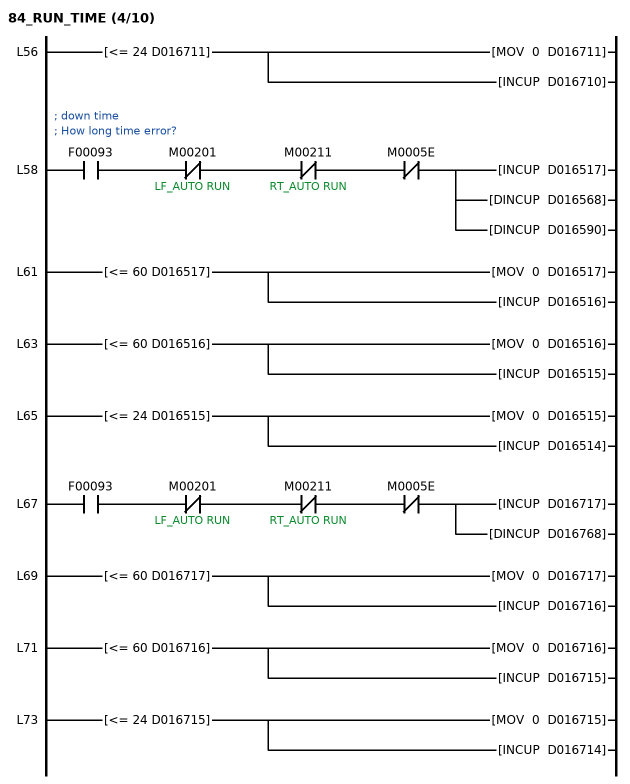
[picture p360: 84_RUN_TIME rungs L56-L73]
; L56
LOAD<=    24 D016711
MOV       0 D016711
INCUP     D016710
; L58
LOAD      F00093
AND NOT   M00201	// LF_AUTO RUN
AND NOT   M00211	// RT_AUTO RUN
AND NOT   M0005E
INCUP     D016517
DINCUP    D016568
DINCUP    D016590
// output comment: down time
// output comment: How long time error?
; L61
LOAD<=    60 D016517
MOV       0 D016517
INCUP     D016516
; L63
LOAD<=    60 D016516
MOV       0 D016516
INCUP     D016515
; L65
LOAD<=    24 D016515
MOV       0 D016515
INCUP     D016514
; L67
LOAD      F00093
AND NOT   M00201	// LF_AUTO RUN
AND NOT   M00211	// RT_AUTO RUN
AND NOT   M0005E
INCUP     D016717
DINCUP    D016768
; L69
LOAD<=    60 D016717
MOV       0 D016717
INCUP     D016716
; L71
LOAD<=    60 D016716
MOV       0 D016716
INCUP     D016715
; L73
LOAD<=    24 D016715
MOV       0 D016715
INCUP     D016714

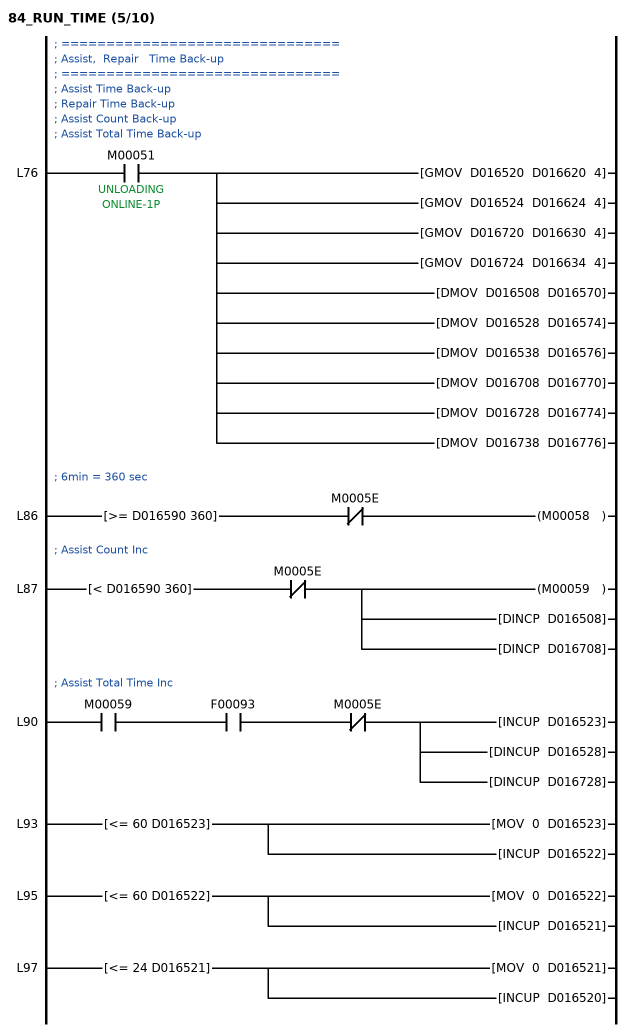
// ===============================
// Assist,  Repair   Time Back-up
// ===============================
; L76
LOAD      M00051	// UNLOADING ONLINE-1P
GMOV      D016520 D016620 4
GMOV      D016524 D016624 4
GMOV      D016720 D016630 4
GMOV      D016724 D016634 4
DMOV      D016508 D016570
DMOV      D016528 D016574
DMOV      D016538 D016576
DMOV      D016708 D016770
DMOV      D016728 D016774
DMOV      D016738 D016776
// output comment: Assist Time Back-up
// output comment: Repair Time Back-up
// output comment: Assist Count Back-up
// output comment: Assist Total Time Back-up
; L86
LOAD>=    D016590 360
AND NOT   M0005E
OUT       M00058
// output comment: 6min = 360 sec
; L87
LOAD<     D016590 360
AND NOT   M0005E
OUT       M00059
DINCP     D016508
DINCP     D016708
// output comment: Assist Count Inc
; L90
LOAD      M00059
AND       F00093
AND NOT   M0005E
INCUP     D016523
DINCUP    D016528
DINCUP    D016728
// output comment: Assist Total Time Inc
; L93
LOAD<=    60 D016523
MOV       0 D016523
INCUP     D016522
; L95
LOAD<=    60 D016522
MOV       0 D016522
INCUP     D016521
; L97
LOAD<=    24 D016521
MOV       0 D016521
INCUP     D016520

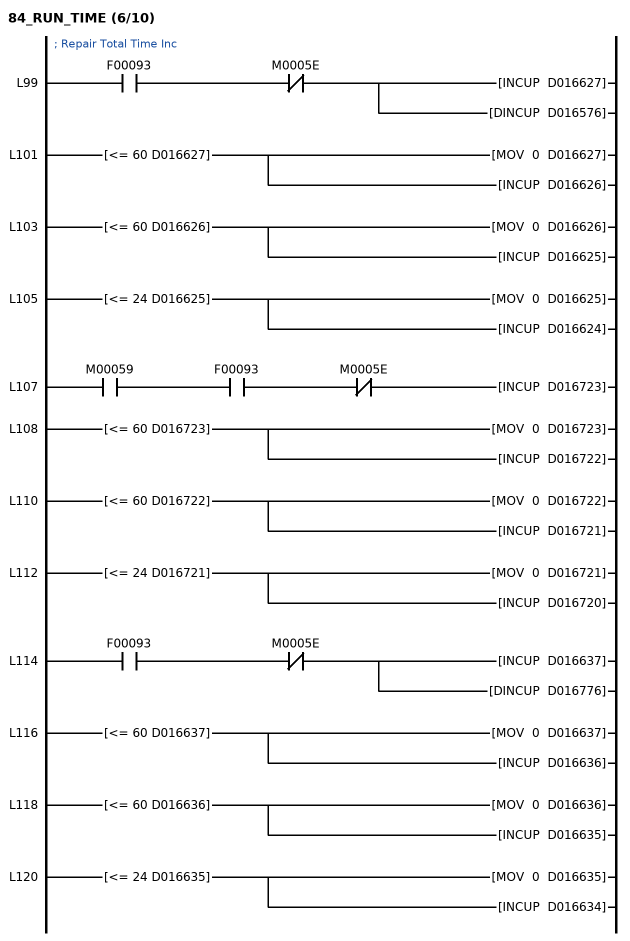
; L99
LOAD      F00093
AND NOT   M0005E
INCUP     D016627
DINCUP    D016576
// output comment: Repair Total Time Inc
; L101
LOAD<=    60 D016627
MOV       0 D016627
INCUP     D016626
; L103
LOAD<=    60 D016626
MOV       0 D016626
INCUP     D016625
; L105
LOAD<=    24 D016625
MOV       0 D016625
INCUP     D016624
; L107
LOAD      M00059
AND       F00093
AND NOT   M0005E
INCUP     D016723
; L108
LOAD<=    60 D016723
MOV       0 D016723
INCUP     D016722
; L110
LOAD<=    60 D016722
MOV       0 D016722
INCUP     D016721
; L112
LOAD<=    24 D016721
MOV       0 D016721
INCUP     D016720
; L114
LOAD      F00093
AND NOT   M0005E
INCUP     D016637
DINCUP    D016776
; L116
LOAD<=    60 D016637
MOV       0 D016637
INCUP     D016636
; L118
LOAD<=    60 D016636
MOV       0 D016636
INCUP     D016635
; L120
LOAD<=    24 D016635
MOV       0 D016635
INCUP     D016634

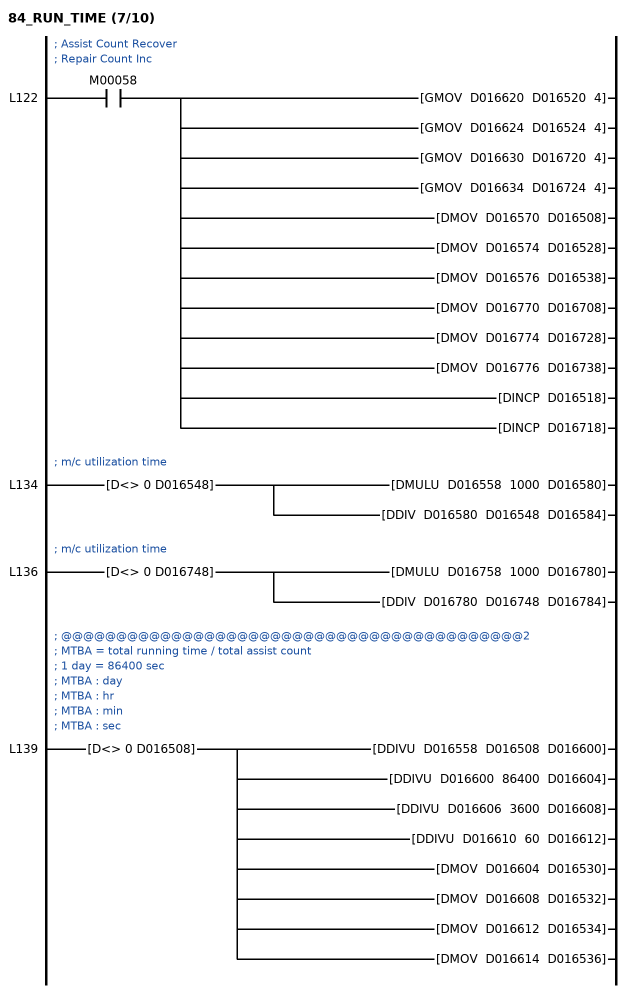
; L122
LOAD      M00058
GMOV      D016620 D016520 4
GMOV      D016624 D016524 4
GMOV      D016630 D016720 4
GMOV      D016634 D016724 4
DMOV      D016570 D016508
DMOV      D016574 D016528
DMOV      D016576 D016538
DMOV      D016770 D016708
DMOV      D016774 D016728
DMOV      D016776 D016738
DINCP     D016518
DINCP     D016718
// output comment: Assist Count Recover
// output comment: Repair Count Inc
; L134
LOADD<>   0 D016548
DMULU     D016558 1000 D016580
DDIV      D016580 D016548 D016584
// output comment: m/c utilization time
; L136
LOADD<>   0 D016748
DMULU     D016758 1000 D016780
DDIV      D016780 D016748 D016784
// output comment: m/c utilization time
// @@@@@@@@@@@@@@@@@@@@@@@@@@@@@@@@@@@@@@@@@@2
; L139
LOADD<>   0 D016508
DDIVU     D016558 D016508 D016600
DDIVU     D016600 86400 D016604
DDIVU     D016606 3600 D016608
DDIVU     D016610 60 D016612
DMOV      D016604 D016530
DMOV      D016608 D016532
DMOV      D016612 D016534
DMOV      D016614 D016536
// output comment: MTBA = total running time / total assist count
// output comment: 1 day = 86400 sec
// output comment: MTBA : day
// output comment: MTBA : hr
// output comment: MTBA : min
// output comment: MTBA : sec

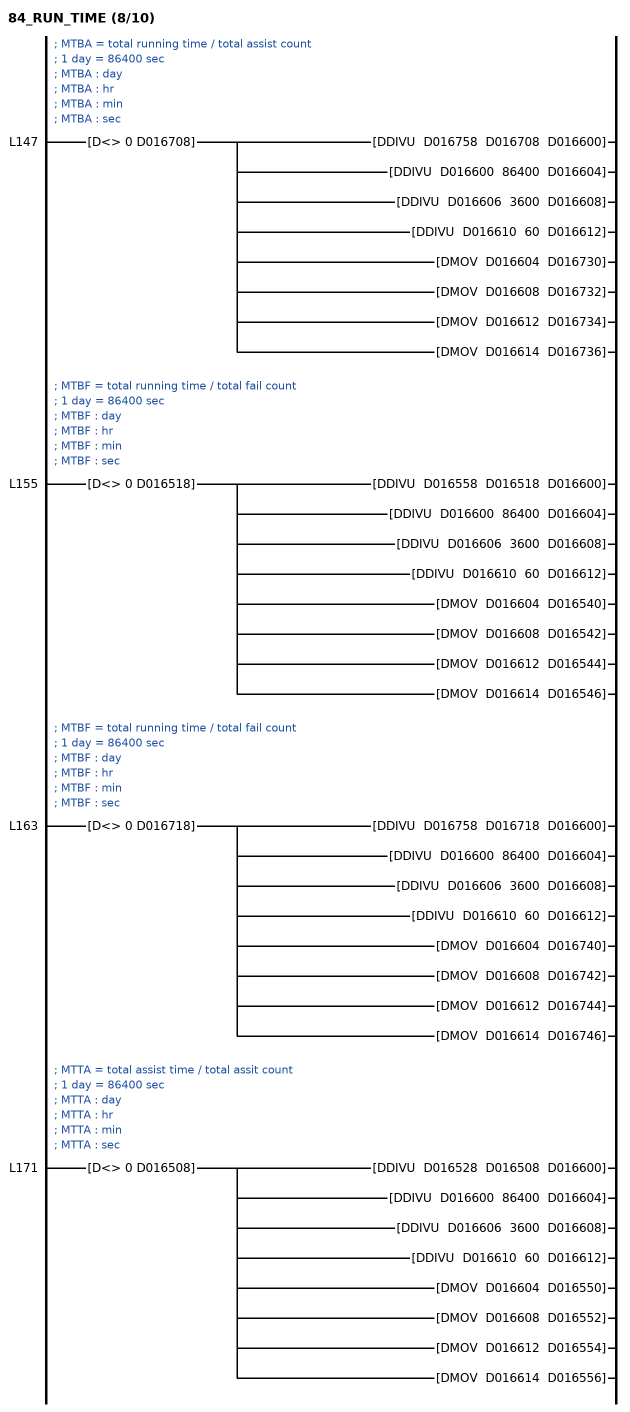
; L147
LOADD<>   0 D016708
DDIVU     D016758 D016708 D016600
DDIVU     D016600 86400 D016604
DDIVU     D016606 3600 D016608
DDIVU     D016610 60 D016612
DMOV      D016604 D016730
DMOV      D016608 D016732
DMOV      D016612 D016734
DMOV      D016614 D016736
// output comment: MTBA = total running time / total assist count
// output comment: 1 day = 86400 sec
// output comment: MTBA : day
// output comment: MTBA : hr
// output comment: MTBA : min
// output comment: MTBA : sec
; L155
LOADD<>   0 D016518
DDIVU     D016558 D016518 D016600
DDIVU     D016600 86400 D016604
DDIVU     D016606 3600 D016608
DDIVU     D016610 60 D016612
DMOV      D016604 D016540
DMOV      D016608 D016542
DMOV      D016612 D016544
DMOV      D016614 D016546
// output comment: MTBF = total running time / total fail count
// output comment: 1 day = 86400 sec
// output comment: MTBF : day
// output comment: MTBF : hr
// output comment: MTBF : min
// output comment: MTBF : sec
; L163
LOADD<>   0 D016718
DDIVU     D016758 D016718 D016600
DDIVU     D016600 86400 D016604
DDIVU     D016606 3600 D016608
DDIVU     D016610 60 D016612
DMOV      D016604 D016740
DMOV      D016608 D016742
DMOV      D016612 D016744
DMOV      D016614 D016746
// output comment: MTBF = total running time / total fail count
// output comment: 1 day = 86400 sec
// output comment: MTBF : day
// output comment: MTBF : hr
// output comment: MTBF : min
// output comment: MTBF : sec
; L171
LOADD<>   0 D016508
DDIVU     D016528 D016508 D016600
DDIVU     D016600 86400 D016604
DDIVU     D016606 3600 D016608
DDIVU     D016610 60 D016612
DMOV      D016604 D016550
DMOV      D016608 D016552
DMOV      D016612 D016554
DMOV      D016614 D016556
// output comment: MTTA = total assist time / total assit count
// output comment: 1 day = 86400 sec
// output comment: MTTA : day
// output comment: MTTA : hr
// output comment: MTTA : min
// output comment: MTTA : sec

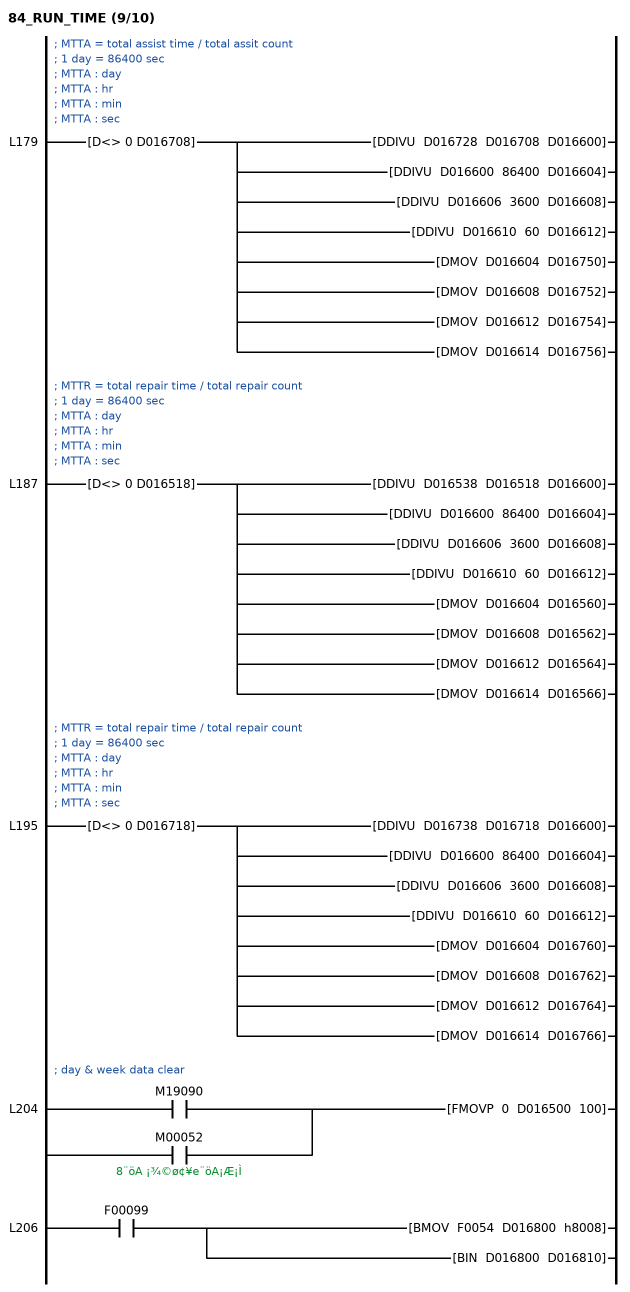
; L179
LOADD<>   0 D016708
DDIVU     D016728 D016708 D016600
DDIVU     D016600 86400 D016604
DDIVU     D016606 3600 D016608
DDIVU     D016610 60 D016612
DMOV      D016604 D016750
DMOV      D016608 D016752
DMOV      D016612 D016754
DMOV      D016614 D016756
// output comment: MTTA = total assist time / total assit count
// output comment: 1 day = 86400 sec
// output comment: MTTA : day
// output comment: MTTA : hr
// output comment: MTTA : min
// output comment: MTTA : sec
; L187
LOADD<>   0 D016518
DDIVU     D016538 D016518 D016600
DDIVU     D016600 86400 D016604
DDIVU     D016606 3600 D016608
DDIVU     D016610 60 D016612
DMOV      D016604 D016560
DMOV      D016608 D016562
DMOV      D016612 D016564
DMOV      D016614 D016566
// output comment: MTTR = total repair time / total repair count
// output comment: 1 day = 86400 sec
// output comment: MTTA : day
// output comment: MTTA : hr
// output comment: MTTA : min
// output comment: MTTA : sec
; L195
LOADD<>   0 D016718
DDIVU     D016738 D016718 D016600
DDIVU     D016600 86400 D016604
DDIVU     D016606 3600 D016608
DDIVU     D016610 60 D016612
DMOV      D016604 D016760
DMOV      D016608 D016762
DMOV      D016612 D016764
DMOV      D016614 D016766
// output comment: MTTR = total repair time / total repair count
// output comment: 1 day = 86400 sec
// output comment: MTTA : day
// output comment: MTTA : hr
// output comment: MTTA : min
// output comment: MTTA : sec
// day & week data clear
; L204
LOAD      M19090
OR        M00052	// 8¨öA ¡¾©ø¢¥e¨öA¡Æ¡Ì
FMOVP     0 D016500 100
; L206
LOAD      F00099
BMOV      F0054 D016800 h8008
BIN       D016800 D016810

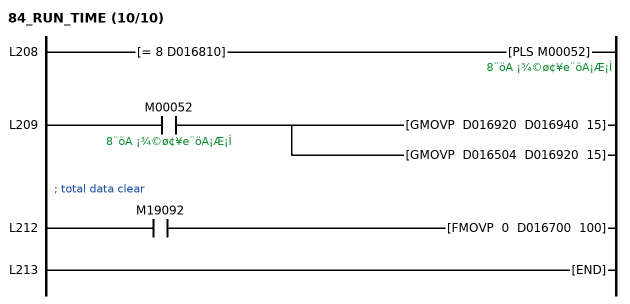
; L208
LOAD=     8 D016810
OUTP      M00052	// 8¨öA ¡¾©ø¢¥e¨öA¡Æ¡Ì
; L209
LOAD      M00052	// 8¨öA ¡¾©ø¢¥e¨öA¡Æ¡Ì
GMOVP     D016920 D016940 15
GMOVP     D016504 D016920 15
// total data clear
; L212
LOAD      M19092
FMOVP     0 D016700 100
; L213
END

PROGRAM 90_ALARM (task: ¨ö¨¬A¥ì CA¡¤I¡¾¡¿¡¤¡Í)

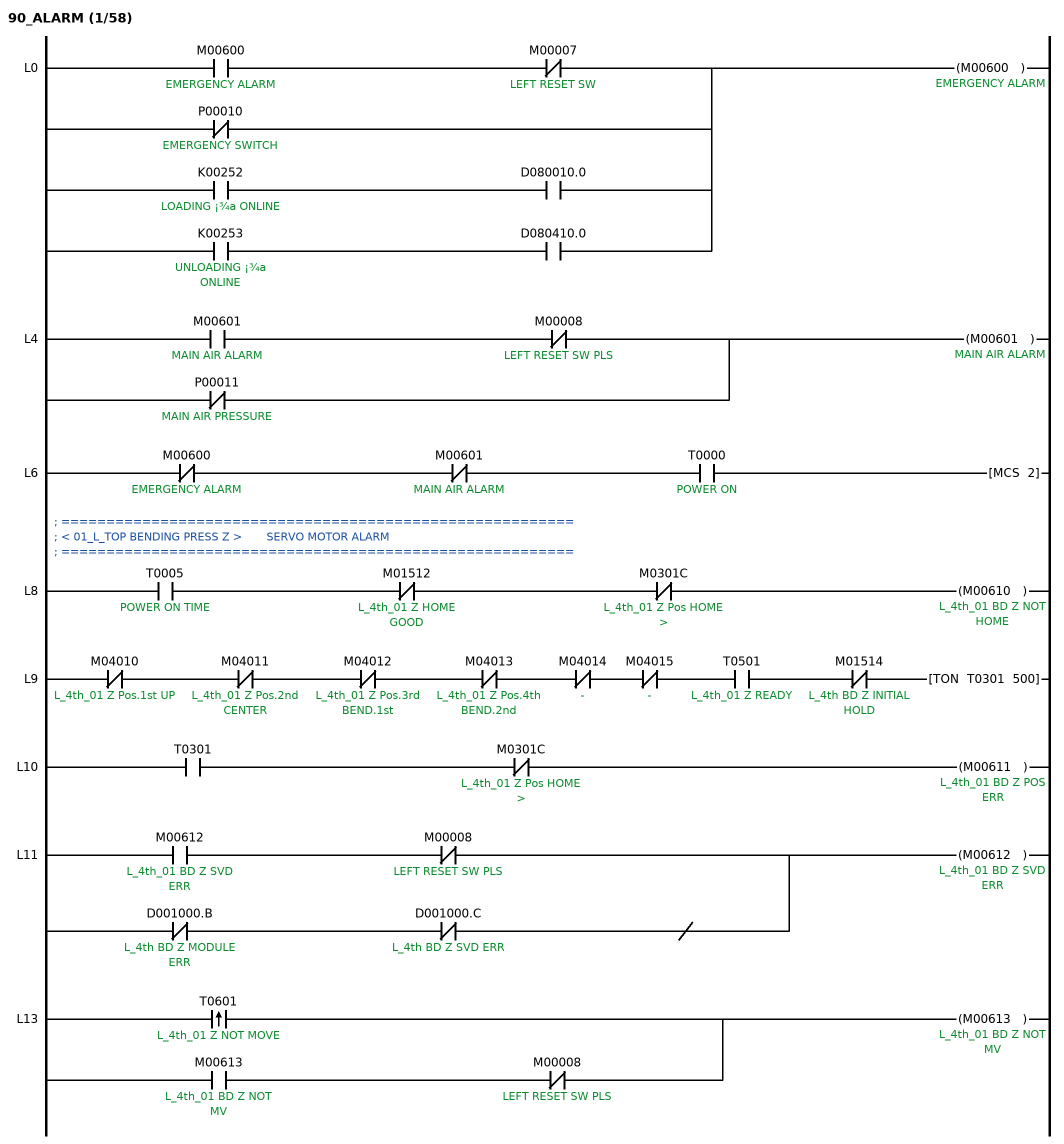
; L0
LOAD      M00600	// EMERGENCY ALARM
AND NOT   M00007	// LEFT RESET SW
OR NOT    P00010	// EMERGENCY SWITCH
LOAD      K00252	// LOADING ¡¾a ONLINE
AND       D080010.0
OR LOAD
LOAD      K00253	// UNLOADING ¡¾a ONLINE
AND       D080410.0
OR LOAD
OUT       M00600	// EMERGENCY ALARM
; L4
LOAD      M00601	// MAIN AIR ALARM
AND NOT   M00008	// LEFT RESET SW PLS
OR NOT    P00011	// MAIN AIR PRESSURE
OUT       M00601	// MAIN AIR ALARM
; L6
LOAD NOT  M00600	// EMERGENCY ALARM
AND NOT   M00601	// MAIN AIR ALARM
AND       T0000	// POWER ON
MCS       2
// =========================================================
// 
//        < 01_L_TOP BENDING PRESS Z >       SERVO MOTOR ALARM
// 
// =========================================================
; L8
LOAD      T0005	// POWER ON TIME
AND NOT   M01512	// L_4th_01 Z HOME GOOD
AND NOT   M0301C	// L_4th_01 Z Pos HOME >
OUT       M00610	// L_4th_01 BD Z NOT HOME
; L9
LOAD NOT  M04010	// L_4th_01 Z Pos.1st UP
AND NOT   M04011	// L_4th_01 Z Pos.2nd CENTER
AND NOT   M04012	// L_4th_01 Z Pos.3rd BEND.1st
AND NOT   M04013	// L_4th_01 Z Pos.4th BEND.2nd
AND NOT   M04014	// -
AND NOT   M04015	// -
AND       T0501	// L_4th_01 Z READY
AND NOT   M01514	// L_4th BD Z INITIAL HOLD
TON       T0301 500
; L10
LOAD      T0301
AND NOT   M0301C	// L_4th_01 Z Pos HOME >
OUT       M00611	// L_4th_01 BD Z POS ERR
; L11
LOAD      M00612	// L_4th_01 BD Z SVD ERR
AND NOT   M00008	// LEFT RESET SW PLS
LOAD NOT  D001000.B	// L_4th BD Z MODULE ERR
AND NOT   D001000.C	// L_4th BD Z SVD ERR
NOT
OR LOAD
OUT       M00612	// L_4th_01 BD Z SVD ERR
; L13
LOADP     T0601	// L_4th_01 Z NOT MOVE
LOAD      M00613	// L_4th_01 BD Z NOT MV
AND NOT   M00008	// LEFT RESET SW PLS
OR LOAD
OUT       M00613	// L_4th_01 BD Z NOT MV

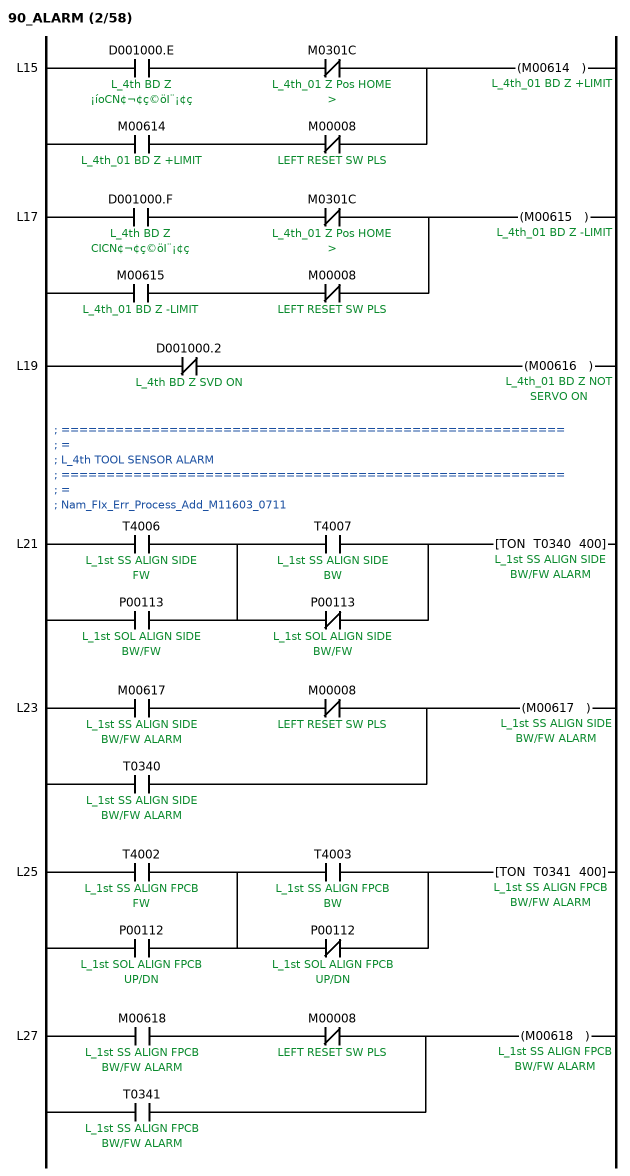
; L15
LOAD      D001000.E	// L_4th BD Z ¡íoCN¢¬¢ç©öI¨¡¢ç
AND NOT   M0301C	// L_4th_01 Z Pos HOME >
LOAD      M00614	// L_4th_01 BD Z +LIMIT
AND NOT   M00008	// LEFT RESET SW PLS
OR LOAD
OUT       M00614	// L_4th_01 BD Z +LIMIT
; L17
LOAD      D001000.F	// L_4th BD Z CICN¢¬¢ç©öI¨¡¢ç
AND NOT   M0301C	// L_4th_01 Z Pos HOME >
LOAD      M00615	// L_4th_01 BD Z -LIMIT
AND NOT   M00008	// LEFT RESET SW PLS
OR LOAD
OUT       M00615	// L_4th_01 BD Z -LIMIT
; L19
LOAD NOT  D001000.2	// L_4th BD Z SVD ON
OUT       M00616	// L_4th_01 BD Z NOT SERVO ON
// =========================================================
// 
//        L_4th TOOL SENSOR ALARM
// 
// =========================================================
; L21
LOAD      T4006	// L_1st SS ALIGN SIDE FW
OR        P00113	// L_1st SOL ALIGN SIDE BW/FW
LOAD      T4007	// L_1st SS ALIGN SIDE BW
OR NOT    P00113	// L_1st SOL ALIGN SIDE BW/FW
AND LOAD
TON       T0340 400	// L_1st SS ALIGN SIDE BW/FW ALARM
// output comment: Nam_FIx_Err_Process_Add_M11603_0711
; L23
LOAD      M00617	// L_1st SS ALIGN SIDE BW/FW ALARM
AND NOT   M00008	// LEFT RESET SW PLS
OR        T0340	// L_1st SS ALIGN SIDE BW/FW ALARM
OUT       M00617	// L_1st SS ALIGN SIDE BW/FW ALARM
; L25
LOAD      T4002	// L_1st SS ALIGN FPCB FW
OR        P00112	// L_1st SOL ALIGN FPCB UP/DN
LOAD      T4003	// L_1st SS ALIGN FPCB BW
OR NOT    P00112	// L_1st SOL ALIGN FPCB UP/DN
AND LOAD
TON       T0341 400	// L_1st SS ALIGN FPCB BW/FW ALARM
; L27
LOAD      M00618	// L_1st SS ALIGN FPCB BW/FW ALARM
AND NOT   M00008	// LEFT RESET SW PLS
OR        T0341	// L_1st SS ALIGN FPCB BW/FW ALARM
OUT       M00618	// L_1st SS ALIGN FPCB BW/FW ALARM

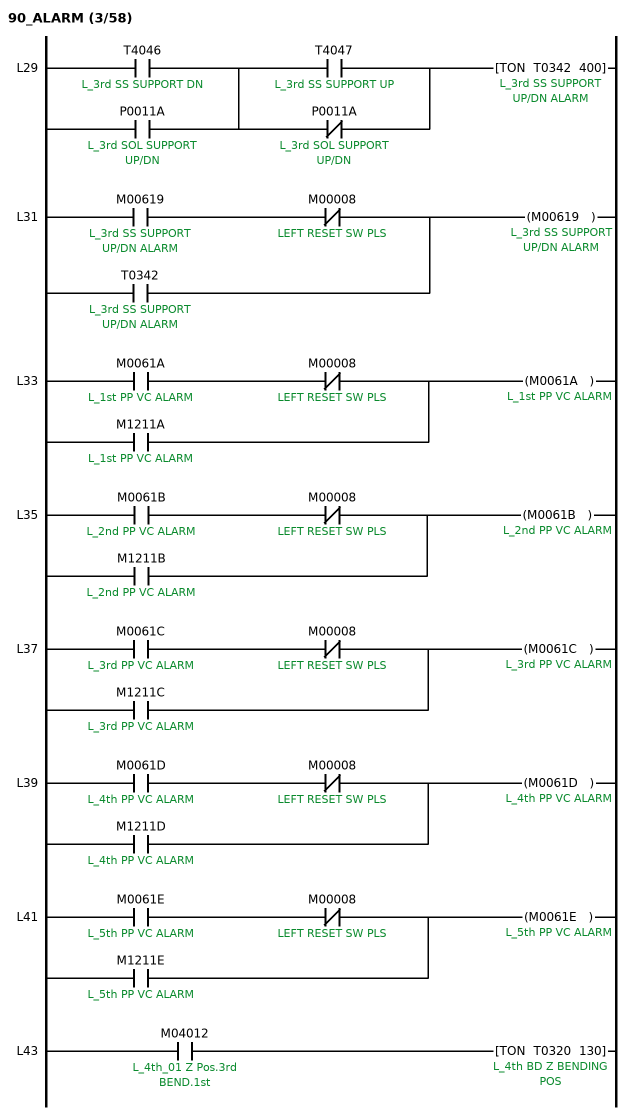
; L29
LOAD      T4046	// L_3rd SS SUPPORT DN
OR        P0011A	// L_3rd SOL SUPPORT UP/DN
LOAD      T4047	// L_3rd SS SUPPORT UP
OR NOT    P0011A	// L_3rd SOL SUPPORT UP/DN
AND LOAD
TON       T0342 400	// L_3rd SS SUPPORT UP/DN ALARM
; L31
LOAD      M00619	// L_3rd SS SUPPORT UP/DN ALARM
AND NOT   M00008	// LEFT RESET SW PLS
OR        T0342	// L_3rd SS SUPPORT UP/DN ALARM
OUT       M00619	// L_3rd SS SUPPORT UP/DN ALARM
; L33
LOAD      M0061A	// L_1st PP VC ALARM
AND NOT   M00008	// LEFT RESET SW PLS
OR        M1211A	// L_1st PP VC ALARM
OUT       M0061A	// L_1st PP VC ALARM
; L35
LOAD      M0061B	// L_2nd PP VC ALARM
AND NOT   M00008	// LEFT RESET SW PLS
OR        M1211B	// L_2nd PP VC ALARM
OUT       M0061B	// L_2nd PP VC ALARM
; L37
LOAD      M0061C	// L_3rd PP VC ALARM
AND NOT   M00008	// LEFT RESET SW PLS
OR        M1211C	// L_3rd PP VC ALARM
OUT       M0061C	// L_3rd PP VC ALARM
; L39
LOAD      M0061D	// L_4th PP VC ALARM
AND NOT   M00008	// LEFT RESET SW PLS
OR        M1211D	// L_4th PP VC ALARM
OUT       M0061D	// L_4th PP VC ALARM
; L41
LOAD      M0061E	// L_5th PP VC ALARM
AND NOT   M00008	// LEFT RESET SW PLS
OR        M1211E	// L_5th PP VC ALARM
OUT       M0061E	// L_5th PP VC ALARM
; L43
LOAD      M04012	// L_4th_01 Z Pos.3rd BEND.1st
TON       T0320 130	// L_4th BD Z BENDING POS

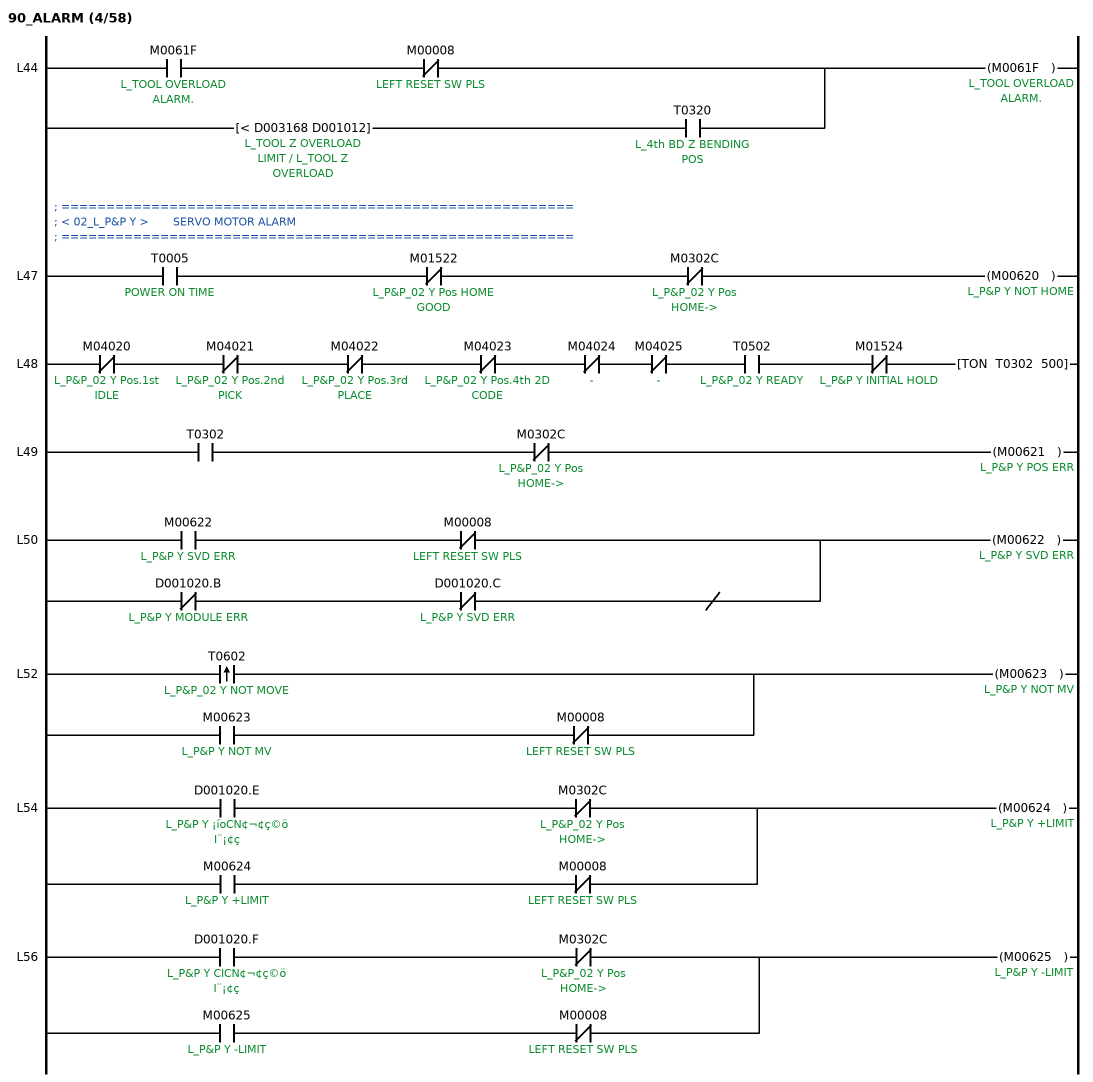
; L44
LOAD      M0061F	// L_TOOL OVERLOAD ALARM.
AND NOT   M00008	// LEFT RESET SW PLS
LOAD<     D003168 D001012	// L_TOOL Z OVERLOAD LIMIT / L_TOOL Z OVERLOAD
AND       T0320	// L_4th BD Z BENDING POS
OR LOAD
OUT       M0061F	// L_TOOL OVERLOAD ALARM.
// =========================================================
// 
//        < 02_L_P&P Y >       SERVO MOTOR ALARM
// 
// =========================================================
; L47
LOAD      T0005	// POWER ON TIME
AND NOT   M01522	// L_P&P_02 Y Pos HOME GOOD
AND NOT   M0302C	// L_P&P_02 Y Pos HOME->
OUT       M00620	// L_P&P Y NOT HOME
; L48
LOAD NOT  M04020	// L_P&P_02 Y Pos.1st IDLE
AND NOT   M04021	// L_P&P_02 Y Pos.2nd PICK
AND NOT   M04022	// L_P&P_02 Y Pos.3rd PLACE
AND NOT   M04023	// L_P&P_02 Y Pos.4th 2D CODE
AND NOT   M04024	// -
AND NOT   M04025	// -
AND       T0502	// L_P&P_02 Y READY
AND NOT   M01524	// L_P&P Y INITIAL HOLD
TON       T0302 500
; L49
LOAD      T0302
AND NOT   M0302C	// L_P&P_02 Y Pos HOME->
OUT       M00621	// L_P&P Y POS ERR
; L50
LOAD      M00622	// L_P&P Y SVD ERR
AND NOT   M00008	// LEFT RESET SW PLS
LOAD NOT  D001020.B	// L_P&P Y MODULE ERR
AND NOT   D001020.C	// L_P&P Y SVD ERR
NOT
OR LOAD
OUT       M00622	// L_P&P Y SVD ERR
; L52
LOADP     T0602	// L_P&P_02 Y NOT MOVE
LOAD      M00623	// L_P&P Y NOT MV
AND NOT   M00008	// LEFT RESET SW PLS
OR LOAD
OUT       M00623	// L_P&P Y NOT MV
; L54
LOAD      D001020.E	// L_P&P Y ¡íoCN¢¬¢ç©öI¨¡¢ç
AND NOT   M0302C	// L_P&P_02 Y Pos HOME->
LOAD      M00624	// L_P&P Y +LIMIT
AND NOT   M00008	// LEFT RESET SW PLS
OR LOAD
OUT       M00624	// L_P&P Y +LIMIT
; L56
LOAD      D001020.F	// L_P&P Y CICN¢¬¢ç©öI¨¡¢ç
AND NOT   M0302C	// L_P&P_02 Y Pos HOME->
LOAD      M00625	// L_P&P Y -LIMIT
AND NOT   M00008	// LEFT RESET SW PLS
OR LOAD
OUT       M00625	// L_P&P Y -LIMIT

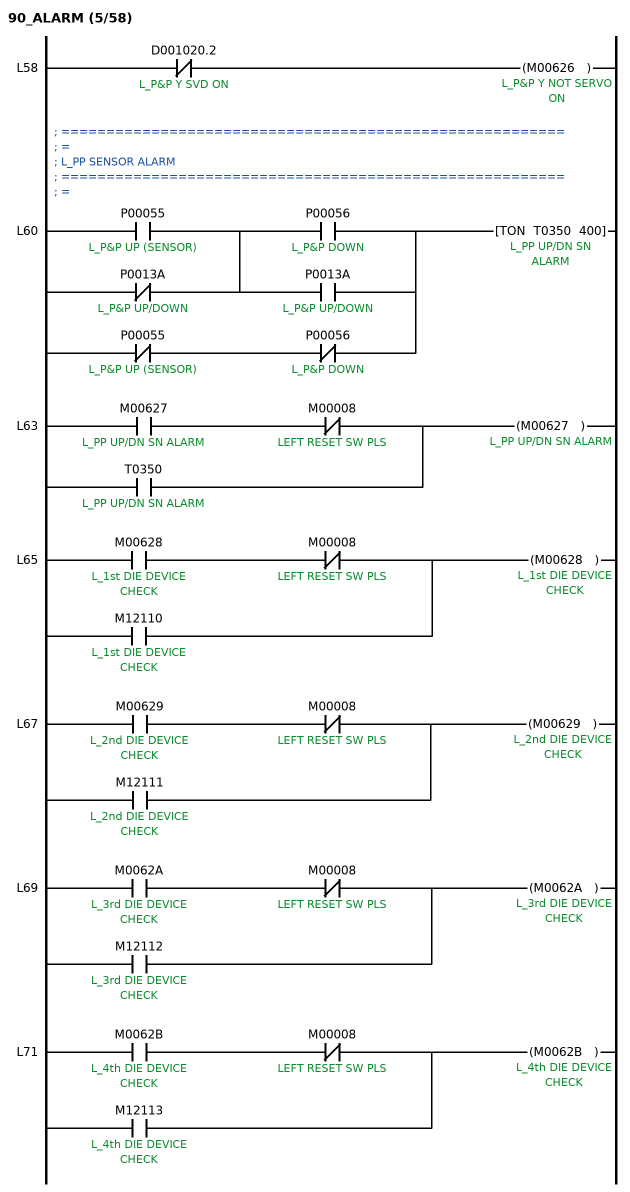
; L58
LOAD NOT  D001020.2	// L_P&P Y SVD ON
OUT       M00626	// L_P&P Y NOT SERVO ON
// =========================================================
// 
//       L_PP SENSOR ALARM
// 
// =========================================================
; L60
LOAD      P00055	// L_P&P UP (SENSOR)
OR NOT    P0013A	// L_P&P UP/DOWN
LOAD      P00056	// L_P&P DOWN
OR        P0013A	// L_P&P UP/DOWN
AND LOAD
LOAD NOT  P00055	// L_P&P UP (SENSOR)
AND NOT   P00056	// L_P&P DOWN
OR LOAD
TON       T0350 400	// L_PP UP/DN SN ALARM
; L63
LOAD      M00627	// L_PP UP/DN SN ALARM
AND NOT   M00008	// LEFT RESET SW PLS
OR        T0350	// L_PP UP/DN SN ALARM
OUT       M00627	// L_PP UP/DN SN ALARM
; L65
LOAD      M00628	// L_1st DIE DEVICE CHECK
AND NOT   M00008	// LEFT RESET SW PLS
OR        M12110	// L_1st DIE DEVICE CHECK
OUT       M00628	// L_1st DIE DEVICE CHECK
; L67
LOAD      M00629	// L_2nd DIE DEVICE CHECK
AND NOT   M00008	// LEFT RESET SW PLS
OR        M12111	// L_2nd DIE DEVICE CHECK
OUT       M00629	// L_2nd DIE DEVICE CHECK
; L69
LOAD      M0062A	// L_3rd DIE DEVICE CHECK
AND NOT   M00008	// LEFT RESET SW PLS
OR        M12112	// L_3rd DIE DEVICE CHECK
OUT       M0062A	// L_3rd DIE DEVICE CHECK
; L71
LOAD      M0062B	// L_4th DIE DEVICE CHECK
AND NOT   M00008	// LEFT RESET SW PLS
OR        M12113	// L_4th DIE DEVICE CHECK
OUT       M0062B	// L_4th DIE DEVICE CHECK

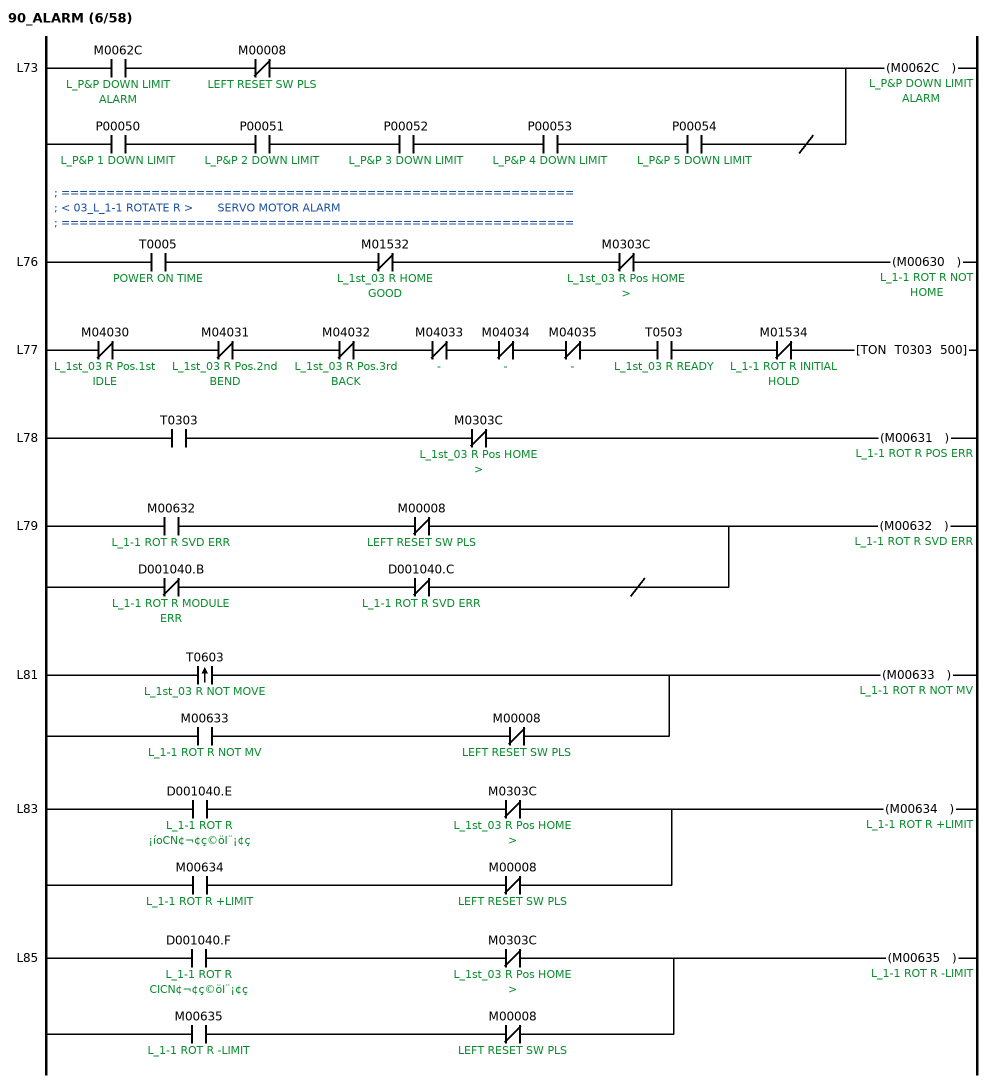
; L73
LOAD      M0062C	// L_P&P DOWN LIMIT ALARM
AND NOT   M00008	// LEFT RESET SW PLS
LOAD      P00050	// L_P&P 1 DOWN LIMIT
AND       P00051	// L_P&P 2 DOWN LIMIT
AND       P00052	// L_P&P 3 DOWN LIMIT
AND       P00053	// L_P&P 4 DOWN LIMIT
AND       P00054	// L_P&P 5 DOWN LIMIT
NOT
OR LOAD
OUT       M0062C	// L_P&P DOWN LIMIT ALARM
// =========================================================
// 
//        < 03_L_1-1 ROTATE R >       SERVO MOTOR ALARM
// 
// =========================================================
; L76
LOAD      T0005	// POWER ON TIME
AND NOT   M01532	// L_1st_03 R HOME GOOD
AND NOT   M0303C	// L_1st_03 R Pos HOME >
OUT       M00630	// L_1-1 ROT R NOT HOME
; L77
LOAD NOT  M04030	// L_1st_03 R Pos.1st IDLE
AND NOT   M04031	// L_1st_03 R Pos.2nd BEND
AND NOT   M04032	// L_1st_03 R Pos.3rd BACK
AND NOT   M04033	// -
AND NOT   M04034	// -
AND NOT   M04035	// -
AND       T0503	// L_1st_03 R READY
AND NOT   M01534	// L_1-1 ROT R INITIAL HOLD
TON       T0303 500
; L78
LOAD      T0303
AND NOT   M0303C	// L_1st_03 R Pos HOME >
OUT       M00631	// L_1-1 ROT R POS ERR
; L79
LOAD      M00632	// L_1-1 ROT R SVD ERR
AND NOT   M00008	// LEFT RESET SW PLS
LOAD NOT  D001040.B	// L_1-1 ROT R MODULE ERR
AND NOT   D001040.C	// L_1-1 ROT R SVD ERR
NOT
OR LOAD
OUT       M00632	// L_1-1 ROT R SVD ERR
; L81
LOADP     T0603	// L_1st_03 R NOT MOVE
LOAD      M00633	// L_1-1 ROT R NOT MV
AND NOT   M00008	// LEFT RESET SW PLS
OR LOAD
OUT       M00633	// L_1-1 ROT R NOT MV
; L83
LOAD      D001040.E	// L_1-1 ROT R ¡íoCN¢¬¢ç©öI¨¡¢ç
AND NOT   M0303C	// L_1st_03 R Pos HOME >
LOAD      M00634	// L_1-1 ROT R +LIMIT
AND NOT   M00008	// LEFT RESET SW PLS
OR LOAD
OUT       M00634	// L_1-1 ROT R +LIMIT
; L85
LOAD      D001040.F	// L_1-1 ROT R CICN¢¬¢ç©öI¨¡¢ç
AND NOT   M0303C	// L_1st_03 R Pos HOME >
LOAD      M00635	// L_1-1 ROT R -LIMIT
AND NOT   M00008	// LEFT RESET SW PLS
OR LOAD
OUT       M00635	// L_1-1 ROT R -LIMIT

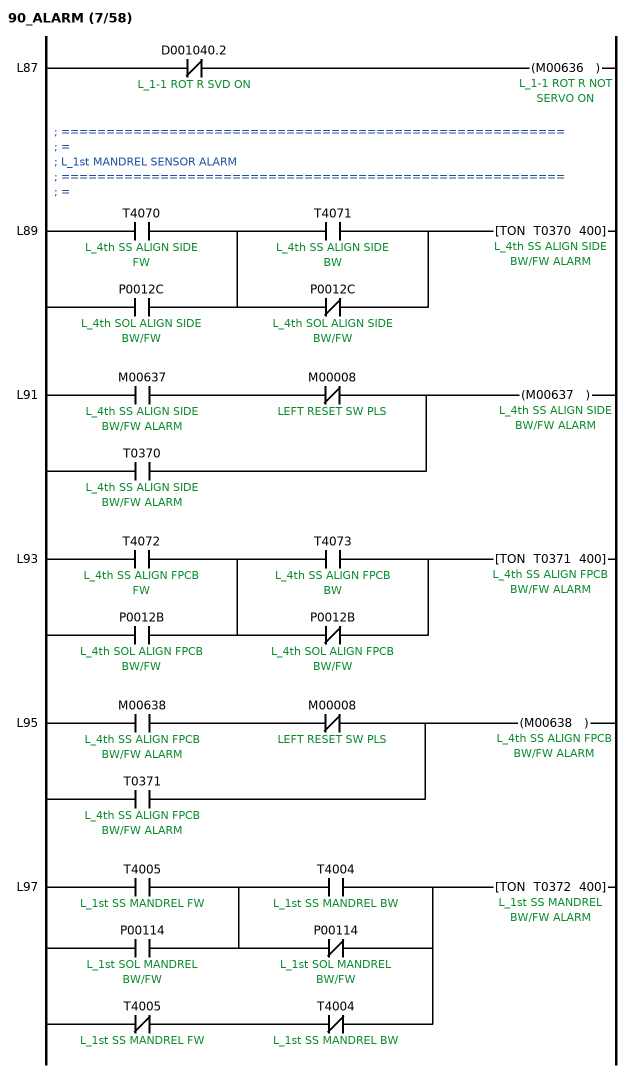
; L87
LOAD NOT  D001040.2	// L_1-1 ROT R SVD ON
OUT       M00636	// L_1-1 ROT R NOT SERVO ON
// =========================================================
// 
//        L_1st MANDREL SENSOR ALARM
// 
// =========================================================
; L89
LOAD      T4070	// L_4th SS ALIGN SIDE FW
OR        P0012C	// L_4th SOL ALIGN SIDE BW/FW
LOAD      T4071	// L_4th SS ALIGN SIDE BW
OR NOT    P0012C	// L_4th SOL ALIGN SIDE BW/FW
AND LOAD
TON       T0370 400	// L_4th SS ALIGN SIDE BW/FW ALARM
; L91
LOAD      M00637	// L_4th SS ALIGN SIDE BW/FW ALARM
AND NOT   M00008	// LEFT RESET SW PLS
OR        T0370	// L_4th SS ALIGN SIDE BW/FW ALARM
OUT       M00637	// L_4th SS ALIGN SIDE BW/FW ALARM
; L93
LOAD      T4072	// L_4th SS ALIGN FPCB FW
OR        P0012B	// L_4th SOL ALIGN FPCB BW/FW
LOAD      T4073	// L_4th SS ALIGN FPCB BW
OR NOT    P0012B	// L_4th SOL ALIGN FPCB BW/FW
AND LOAD
TON       T0371 400	// L_4th SS ALIGN FPCB BW/FW ALARM
; L95
LOAD      M00638	// L_4th SS ALIGN FPCB BW/FW ALARM
AND NOT   M00008	// LEFT RESET SW PLS
OR        T0371	// L_4th SS ALIGN FPCB BW/FW ALARM
OUT       M00638	// L_4th SS ALIGN FPCB BW/FW ALARM
; L97
LOAD      T4005	// L_1st SS MANDREL FW
OR        P00114	// L_1st SOL MANDREL BW/FW
LOAD      T4004	// L_1st SS MANDREL BW
OR NOT    P00114	// L_1st SOL MANDREL BW/FW
AND LOAD
LOAD NOT  T4005	// L_1st SS MANDREL FW
AND NOT   T4004	// L_1st SS MANDREL BW
OR LOAD
TON       T0372 400	// L_1st SS MANDREL BW/FW ALARM

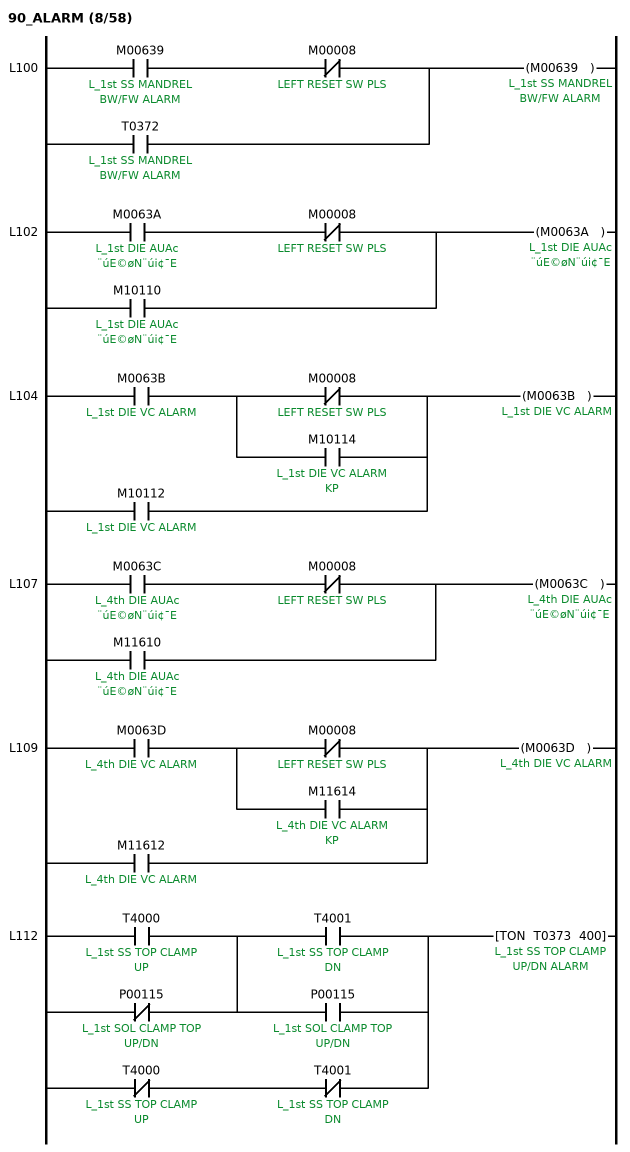
; L100
LOAD      M00639	// L_1st SS MANDREL BW/FW ALARM
AND NOT   M00008	// LEFT RESET SW PLS
OR        T0372	// L_1st SS MANDREL BW/FW ALARM
OUT       M00639	// L_1st SS MANDREL BW/FW ALARM
; L102
LOAD      M0063A	// L_1st DIE AUAc ¨úE©øN¨úi¢¯E
AND NOT   M00008	// LEFT RESET SW PLS
OR        M10110	// L_1st DIE AUAc ¨úE©øN¨úi¢¯E
OUT       M0063A	// L_1st DIE AUAc ¨úE©øN¨úi¢¯E
; L104
LOAD      M0063B	// L_1st DIE VC ALARM
LOAD NOT  M00008	// LEFT RESET SW PLS
OR        M10114	// L_1st DIE VC ALARM KP
AND LOAD
OR        M10112	// L_1st DIE VC ALARM
OUT       M0063B	// L_1st DIE VC ALARM
; L107
LOAD      M0063C	// L_4th DIE AUAc ¨úE©øN¨úi¢¯E
AND NOT   M00008	// LEFT RESET SW PLS
OR        M11610	// L_4th DIE AUAc ¨úE©øN¨úi¢¯E
OUT       M0063C	// L_4th DIE AUAc ¨úE©øN¨úi¢¯E
; L109
LOAD      M0063D	// L_4th DIE VC ALARM
LOAD NOT  M00008	// LEFT RESET SW PLS
OR        M11614	// L_4th DIE VC ALARM KP
AND LOAD
OR        M11612	// L_4th DIE VC ALARM
OUT       M0063D	// L_4th DIE VC ALARM
; L112
LOAD      T4000	// L_1st SS TOP CLAMP    UP
OR NOT    P00115	// L_1st SOL CLAMP TOP UP/DN
LOAD      T4001	// L_1st SS TOP CLAMP    DN
OR        P00115	// L_1st SOL CLAMP TOP UP/DN
AND LOAD
LOAD NOT  T4000	// L_1st SS TOP CLAMP    UP
AND NOT   T4001	// L_1st SS TOP CLAMP    DN
OR LOAD
TON       T0373 400	// L_1st SS TOP CLAMP UP/DN ALARM

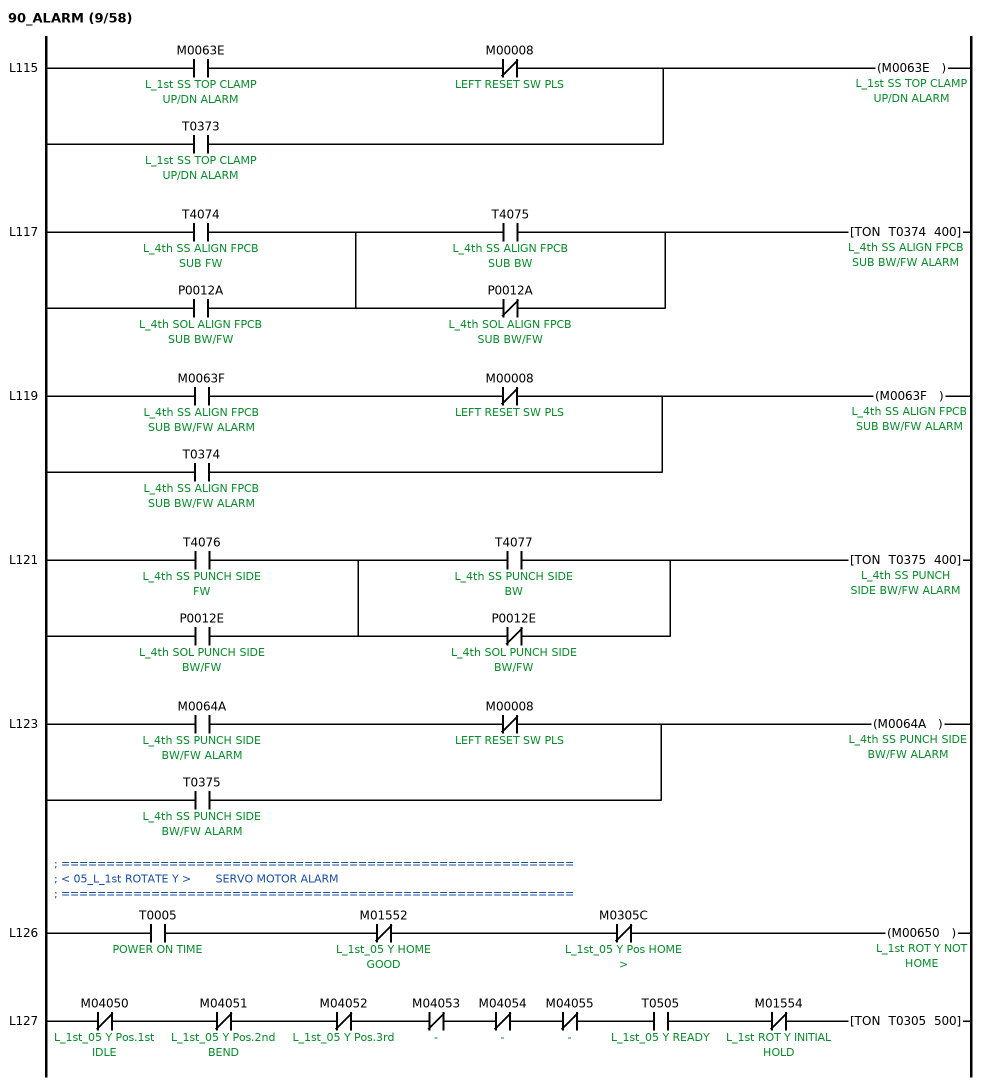
; L115
LOAD      M0063E	// L_1st SS TOP CLAMP UP/DN ALARM
AND NOT   M00008	// LEFT RESET SW PLS
OR        T0373	// L_1st SS TOP CLAMP UP/DN ALARM
OUT       M0063E	// L_1st SS TOP CLAMP UP/DN ALARM
; L117
LOAD      T4074	// L_4th SS ALIGN FPCB SUB FW
OR        P0012A	// L_4th SOL ALIGN FPCB SUB BW/FW
LOAD      T4075	// L_4th SS ALIGN FPCB SUB BW
OR NOT    P0012A	// L_4th SOL ALIGN FPCB SUB BW/FW
AND LOAD
TON       T0374 400	// L_4th SS ALIGN FPCB SUB BW/FW ALARM
; L119
LOAD      M0063F	// L_4th SS ALIGN FPCB SUB BW/FW ALARM
AND NOT   M00008	// LEFT RESET SW PLS
OR        T0374	// L_4th SS ALIGN FPCB SUB BW/FW ALARM
OUT       M0063F	// L_4th SS ALIGN FPCB SUB BW/FW ALARM
; L121
LOAD      T4076	// L_4th SS PUNCH SIDE FW
OR        P0012E	// L_4th SOL PUNCH SIDE BW/FW
LOAD      T4077	// L_4th SS PUNCH SIDE BW
OR NOT    P0012E	// L_4th SOL PUNCH SIDE BW/FW
AND LOAD
TON       T0375 400	// L_4th SS PUNCH SIDE BW/FW ALARM
; L123
LOAD      M0064A	// L_4th SS PUNCH SIDE BW/FW ALARM
AND NOT   M00008	// LEFT RESET SW PLS
OR        T0375	// L_4th SS PUNCH SIDE BW/FW ALARM
OUT       M0064A	// L_4th SS PUNCH SIDE BW/FW ALARM
// =========================================================
// 
//        < 05_L_1st ROTATE Y >       SERVO MOTOR ALARM
// 
// =========================================================
; L126
LOAD      T0005	// POWER ON TIME
AND NOT   M01552	// L_1st_05 Y HOME GOOD
AND NOT   M0305C	// L_1st_05 Y Pos HOME >
OUT       M00650	// L_1st ROT Y NOT HOME
; L127
LOAD NOT  M04050	// L_1st_05 Y Pos.1st IDLE
AND NOT   M04051	// L_1st_05 Y Pos.2nd BEND
AND NOT   M04052	// L_1st_05 Y Pos.3rd
AND NOT   M04053	// -
AND NOT   M04054	// -
AND NOT   M04055	// -
AND       T0505	// L_1st_05 Y READY
AND NOT   M01554	// L_1st ROT Y INITIAL HOLD
TON       T0305 500

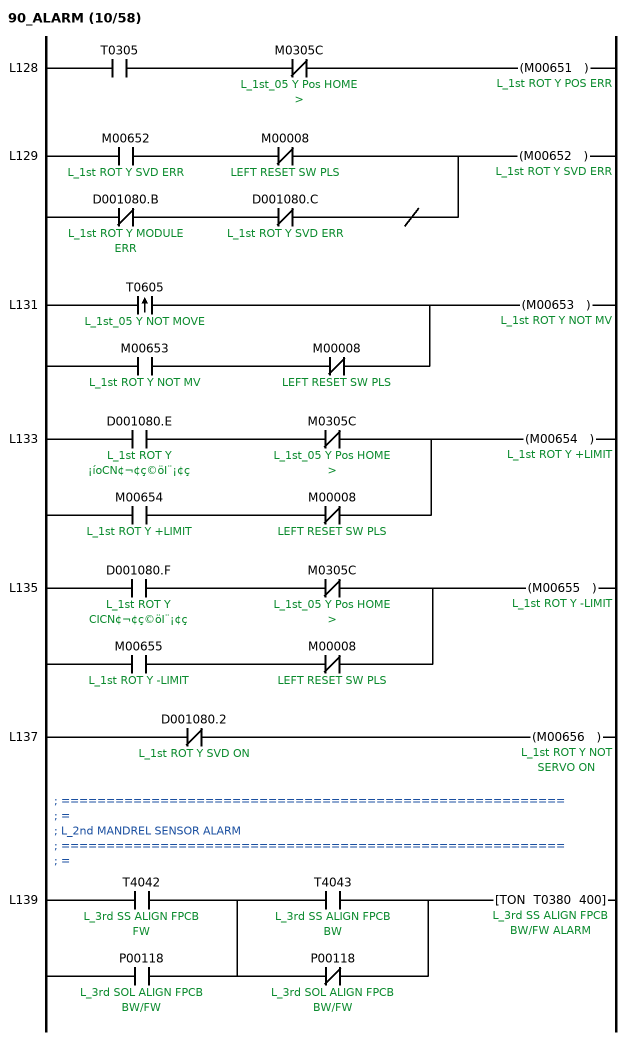
; L128
LOAD      T0305
AND NOT   M0305C	// L_1st_05 Y Pos HOME >
OUT       M00651	// L_1st ROT Y POS ERR
; L129
LOAD      M00652	// L_1st ROT Y SVD ERR
AND NOT   M00008	// LEFT RESET SW PLS
LOAD NOT  D001080.B	// L_1st ROT Y MODULE ERR
AND NOT   D001080.C	// L_1st ROT Y SVD ERR
NOT
OR LOAD
OUT       M00652	// L_1st ROT Y SVD ERR
; L131
LOADP     T0605	// L_1st_05 Y NOT MOVE
LOAD      M00653	// L_1st ROT Y NOT MV
AND NOT   M00008	// LEFT RESET SW PLS
OR LOAD
OUT       M00653	// L_1st ROT Y NOT MV
; L133
LOAD      D001080.E	// L_1st ROT Y ¡íoCN¢¬¢ç©öI¨¡¢ç
AND NOT   M0305C	// L_1st_05 Y Pos HOME >
LOAD      M00654	// L_1st ROT Y +LIMIT
AND NOT   M00008	// LEFT RESET SW PLS
OR LOAD
OUT       M00654	// L_1st ROT Y +LIMIT
; L135
LOAD      D001080.F	// L_1st ROT Y CICN¢¬¢ç©öI¨¡¢ç
AND NOT   M0305C	// L_1st_05 Y Pos HOME >
LOAD      M00655	// L_1st ROT Y -LIMIT
AND NOT   M00008	// LEFT RESET SW PLS
OR LOAD
OUT       M00655	// L_1st ROT Y -LIMIT
; L137
LOAD NOT  D001080.2	// L_1st ROT Y SVD ON
OUT       M00656	// L_1st ROT Y NOT SERVO ON
// =========================================================
// 
//        L_2nd MANDREL SENSOR ALARM
// 
// =========================================================
; L139
LOAD      T4042	// L_3rd SS ALIGN FPCB FW
OR        P00118	// L_3rd SOL ALIGN FPCB BW/FW
LOAD      T4043	// L_3rd SS ALIGN FPCB BW
OR NOT    P00118	// L_3rd SOL ALIGN FPCB BW/FW
AND LOAD
TON       T0380 400	// L_3rd SS ALIGN FPCB BW/FW ALARM

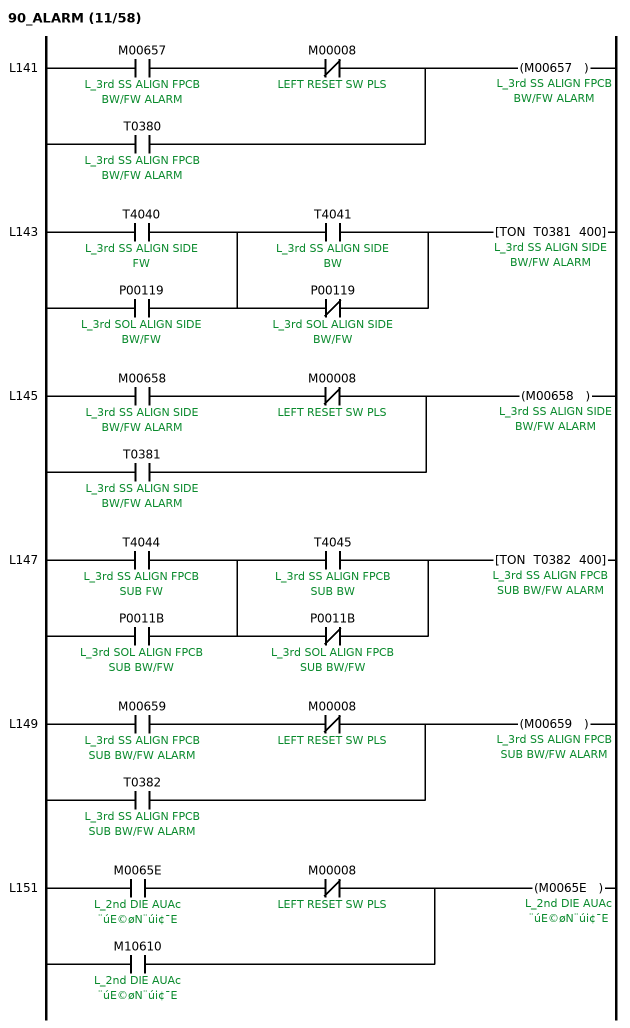
; L141
LOAD      M00657	// L_3rd SS ALIGN FPCB BW/FW ALARM
AND NOT   M00008	// LEFT RESET SW PLS
OR        T0380	// L_3rd SS ALIGN FPCB BW/FW ALARM
OUT       M00657	// L_3rd SS ALIGN FPCB BW/FW ALARM
; L143
LOAD      T4040	// L_3rd SS ALIGN SIDE FW
OR        P00119	// L_3rd SOL ALIGN SIDE BW/FW
LOAD      T4041	// L_3rd SS ALIGN SIDE BW
OR NOT    P00119	// L_3rd SOL ALIGN SIDE BW/FW
AND LOAD
TON       T0381 400	// L_3rd SS ALIGN SIDE BW/FW ALARM
; L145
LOAD      M00658	// L_3rd SS ALIGN SIDE BW/FW ALARM
AND NOT   M00008	// LEFT RESET SW PLS
OR        T0381	// L_3rd SS ALIGN SIDE BW/FW ALARM
OUT       M00658	// L_3rd SS ALIGN SIDE BW/FW ALARM
; L147
LOAD      T4044	// L_3rd SS ALIGN FPCB SUB FW
OR        P0011B	// L_3rd SOL ALIGN FPCB SUB BW/FW
LOAD      T4045	// L_3rd SS ALIGN FPCB SUB BW
OR NOT    P0011B	// L_3rd SOL ALIGN FPCB SUB BW/FW
AND LOAD
TON       T0382 400	// L_3rd SS ALIGN FPCB SUB BW/FW ALARM
; L149
LOAD      M00659	// L_3rd SS ALIGN FPCB SUB BW/FW ALARM
AND NOT   M00008	// LEFT RESET SW PLS
OR        T0382	// L_3rd SS ALIGN FPCB SUB BW/FW ALARM
OUT       M00659	// L_3rd SS ALIGN FPCB SUB BW/FW ALARM
; L151
LOAD      M0065E	// L_2nd DIE AUAc ¨úE©øN¨úi¢¯E
AND NOT   M00008	// LEFT RESET SW PLS
OR        M10610	// L_2nd DIE AUAc ¨úE©øN¨úi¢¯E
OUT       M0065E	// L_2nd DIE AUAc ¨úE©øN¨úi¢¯E

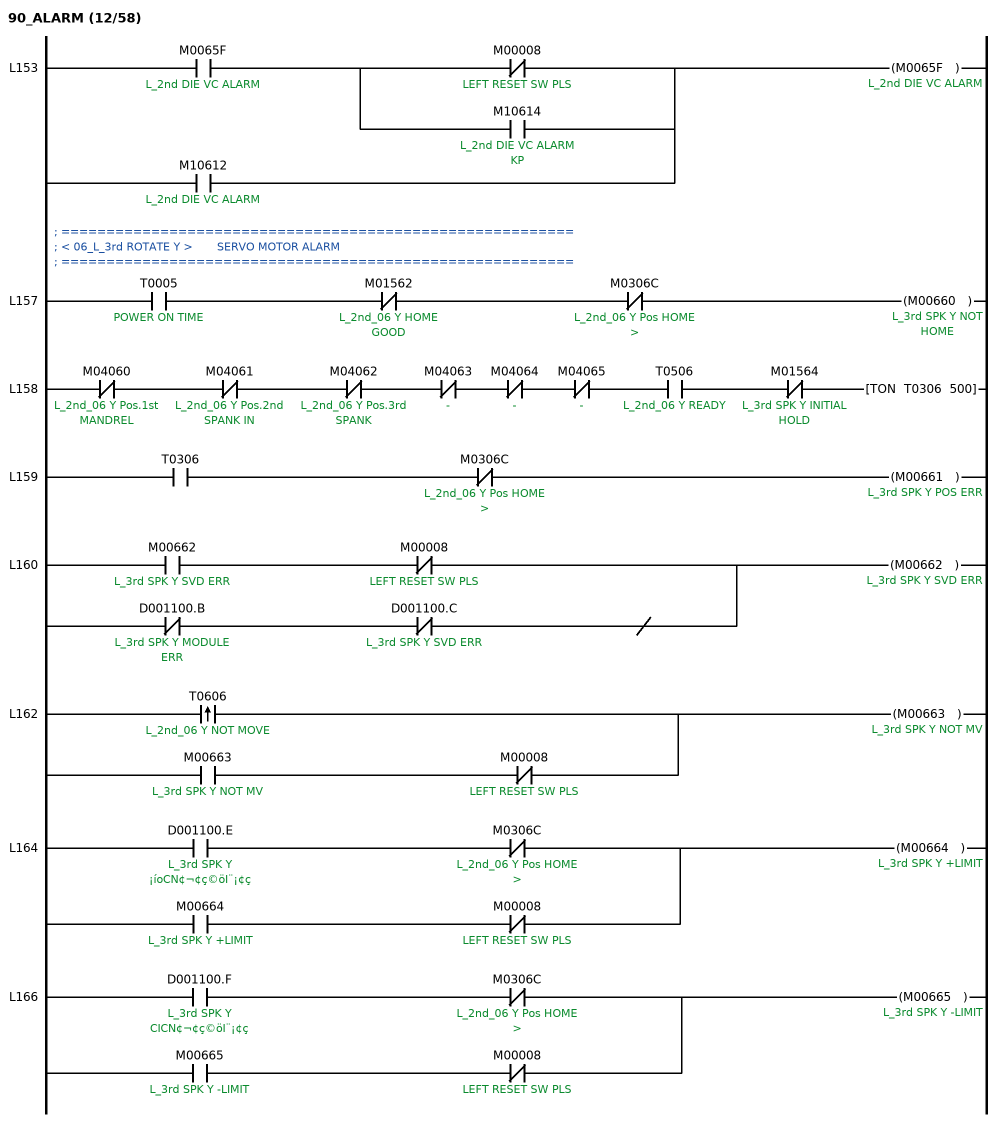
; L153
LOAD      M0065F	// L_2nd DIE VC ALARM
LOAD NOT  M00008	// LEFT RESET SW PLS
OR        M10614	// L_2nd DIE VC ALARM KP
AND LOAD
OR        M10612	// L_2nd DIE VC ALARM
OUT       M0065F	// L_2nd DIE VC ALARM
// =========================================================
// 
//        < 06_L_3rd ROTATE Y >       SERVO MOTOR ALARM
// 
// =========================================================
; L157
LOAD      T0005	// POWER ON TIME
AND NOT   M01562	// L_2nd_06 Y HOME GOOD
AND NOT   M0306C	// L_2nd_06 Y Pos HOME >
OUT       M00660	// L_3rd SPK Y NOT HOME
; L158
LOAD NOT  M04060	// L_2nd_06 Y Pos.1st MANDREL
AND NOT   M04061	// L_2nd_06 Y Pos.2nd SPANK IN
AND NOT   M04062	// L_2nd_06 Y Pos.3rd SPANK
AND NOT   M04063	// -
AND NOT   M04064	// -
AND NOT   M04065	// -
AND       T0506	// L_2nd_06 Y READY
AND NOT   M01564	// L_3rd SPK Y INITIAL HOLD
TON       T0306 500
; L159
LOAD      T0306
AND NOT   M0306C	// L_2nd_06 Y Pos HOME >
OUT       M00661	// L_3rd SPK Y POS ERR
; L160
LOAD      M00662	// L_3rd SPK Y SVD ERR
AND NOT   M00008	// LEFT RESET SW PLS
LOAD NOT  D001100.B	// L_3rd SPK Y MODULE ERR
AND NOT   D001100.C	// L_3rd SPK Y SVD ERR
NOT
OR LOAD
OUT       M00662	// L_3rd SPK Y SVD ERR
; L162
LOADP     T0606	// L_2nd_06 Y NOT MOVE
LOAD      M00663	// L_3rd SPK Y NOT MV
AND NOT   M00008	// LEFT RESET SW PLS
OR LOAD
OUT       M00663	// L_3rd SPK Y NOT MV
; L164
LOAD      D001100.E	// L_3rd SPK Y ¡íoCN¢¬¢ç©öI¨¡¢ç
AND NOT   M0306C	// L_2nd_06 Y Pos HOME >
LOAD      M00664	// L_3rd SPK Y +LIMIT
AND NOT   M00008	// LEFT RESET SW PLS
OR LOAD
OUT       M00664	// L_3rd SPK Y +LIMIT
; L166
LOAD      D001100.F	// L_3rd SPK Y CICN¢¬¢ç©öI¨¡¢ç
AND NOT   M0306C	// L_2nd_06 Y Pos HOME >
LOAD      M00665	// L_3rd SPK Y -LIMIT
AND NOT   M00008	// LEFT RESET SW PLS
OR LOAD
OUT       M00665	// L_3rd SPK Y -LIMIT

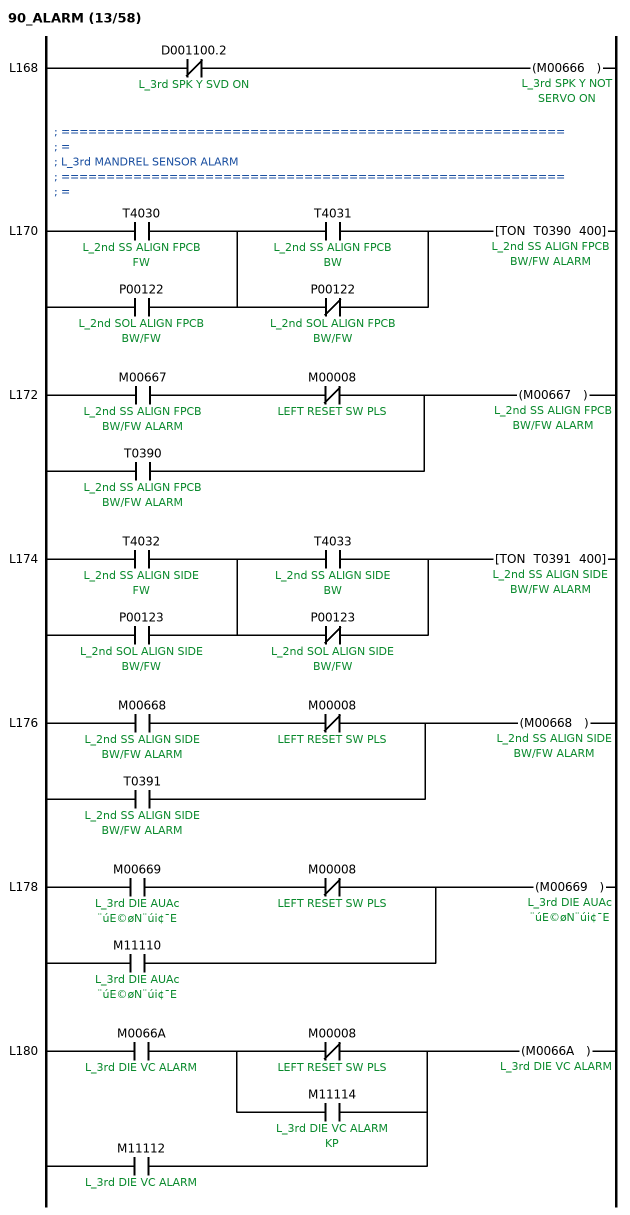
; L168
LOAD NOT  D001100.2	// L_3rd SPK Y SVD ON
OUT       M00666	// L_3rd SPK Y NOT SERVO ON
// =========================================================
// 
//        L_3rd MANDREL SENSOR ALARM
// 
// =========================================================
; L170
LOAD      T4030	// L_2nd SS ALIGN FPCB FW
OR        P00122	// L_2nd SOL ALIGN FPCB BW/FW
LOAD      T4031	// L_2nd SS ALIGN FPCB BW
OR NOT    P00122	// L_2nd SOL ALIGN FPCB BW/FW
AND LOAD
TON       T0390 400	// L_2nd SS ALIGN FPCB BW/FW ALARM
; L172
LOAD      M00667	// L_2nd SS ALIGN FPCB BW/FW ALARM
AND NOT   M00008	// LEFT RESET SW PLS
OR        T0390	// L_2nd SS ALIGN FPCB BW/FW ALARM
OUT       M00667	// L_2nd SS ALIGN FPCB BW/FW ALARM
; L174
LOAD      T4032	// L_2nd SS ALIGN SIDE FW
OR        P00123	// L_2nd SOL ALIGN SIDE BW/FW
LOAD      T4033	// L_2nd SS ALIGN SIDE BW
OR NOT    P00123	// L_2nd SOL ALIGN SIDE BW/FW
AND LOAD
TON       T0391 400	// L_2nd SS ALIGN SIDE BW/FW ALARM
; L176
LOAD      M00668	// L_2nd SS ALIGN SIDE BW/FW ALARM
AND NOT   M00008	// LEFT RESET SW PLS
OR        T0391	// L_2nd SS ALIGN SIDE BW/FW ALARM
OUT       M00668	// L_2nd SS ALIGN SIDE BW/FW ALARM
; L178
LOAD      M00669	// L_3rd DIE AUAc ¨úE©øN¨úi¢¯E
AND NOT   M00008	// LEFT RESET SW PLS
OR        M11110	// L_3rd DIE AUAc ¨úE©øN¨úi¢¯E
OUT       M00669	// L_3rd DIE AUAc ¨úE©øN¨úi¢¯E
; L180
LOAD      M0066A	// L_3rd DIE VC ALARM
LOAD NOT  M00008	// LEFT RESET SW PLS
OR        M11114	// L_3rd DIE VC ALARM KP
AND LOAD
OR        M11112	// L_3rd DIE VC ALARM
OUT       M0066A	// L_3rd DIE VC ALARM

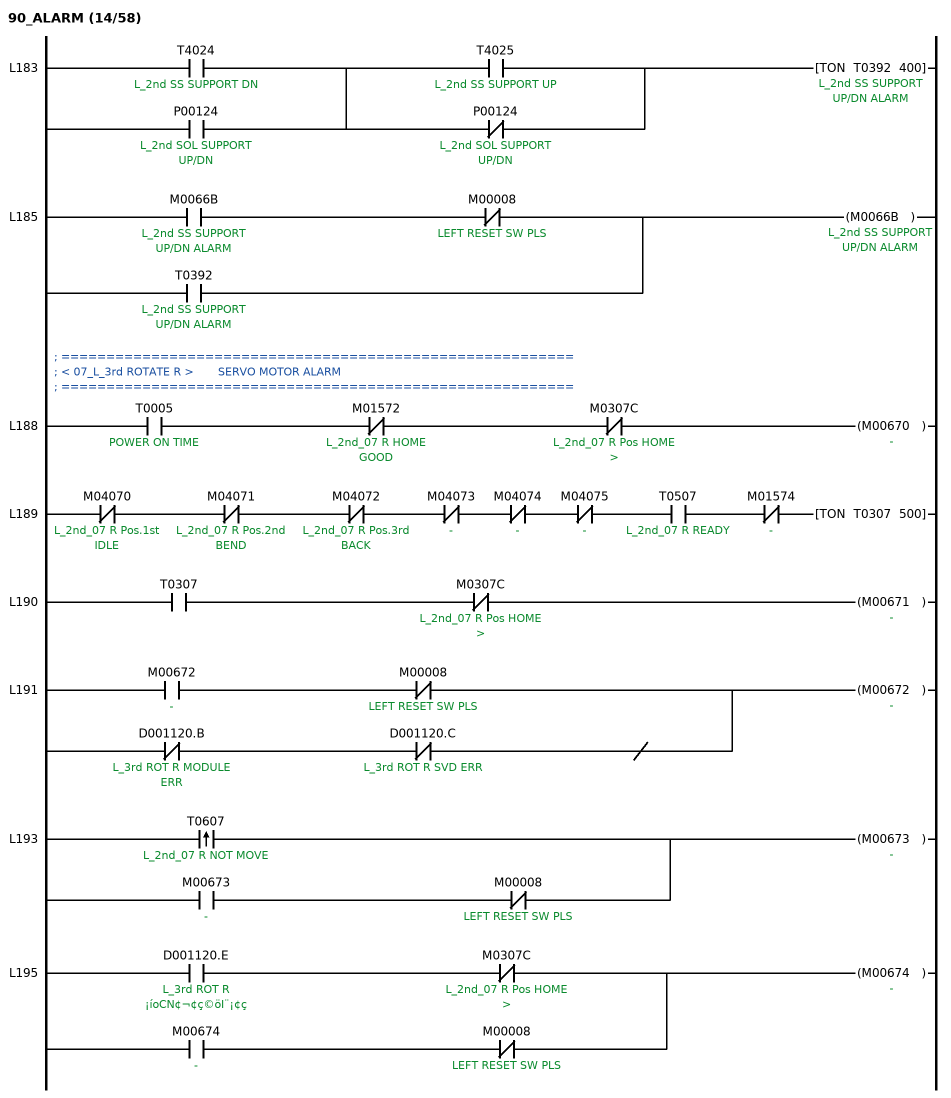
; L183
LOAD      T4024	// L_2nd SS SUPPORT DN
OR        P00124	// L_2nd SOL SUPPORT UP/DN
LOAD      T4025	// L_2nd SS SUPPORT UP
OR NOT    P00124	// L_2nd SOL SUPPORT UP/DN
AND LOAD
TON       T0392 400	// L_2nd SS SUPPORT UP/DN ALARM
; L185
LOAD      M0066B	// L_2nd SS SUPPORT UP/DN ALARM
AND NOT   M00008	// LEFT RESET SW PLS
OR        T0392	// L_2nd SS SUPPORT UP/DN ALARM
OUT       M0066B	// L_2nd SS SUPPORT UP/DN ALARM
// =========================================================
// 
//        < 07_L_3rd ROTATE R >       SERVO MOTOR ALARM
// 
// =========================================================
; L188
LOAD      T0005	// POWER ON TIME
AND NOT   M01572	// L_2nd_07 R HOME GOOD
AND NOT   M0307C	// L_2nd_07 R Pos HOME >
OUT       M00670	// -
; L189
LOAD NOT  M04070	// L_2nd_07 R Pos.1st IDLE
AND NOT   M04071	// L_2nd_07 R Pos.2nd BEND
AND NOT   M04072	// L_2nd_07 R Pos.3rd BACK
AND NOT   M04073	// -
AND NOT   M04074	// -
AND NOT   M04075	// -
AND       T0507	// L_2nd_07 R READY
AND NOT   M01574	// -
TON       T0307 500
; L190
LOAD      T0307
AND NOT   M0307C	// L_2nd_07 R Pos HOME >
OUT       M00671	// -
; L191
LOAD      M00672	// -
AND NOT   M00008	// LEFT RESET SW PLS
LOAD NOT  D001120.B	// L_3rd ROT R MODULE ERR
AND NOT   D001120.C	// L_3rd ROT R SVD ERR
NOT
OR LOAD
OUT       M00672	// -
; L193
LOADP     T0607	// L_2nd_07 R NOT MOVE
LOAD      M00673	// -
AND NOT   M00008	// LEFT RESET SW PLS
OR LOAD
OUT       M00673	// -
; L195
LOAD      D001120.E	// L_3rd ROT R ¡íoCN¢¬¢ç©öI¨¡¢ç
AND NOT   M0307C	// L_2nd_07 R Pos HOME >
LOAD      M00674	// -
AND NOT   M00008	// LEFT RESET SW PLS
OR LOAD
OUT       M00674	// -

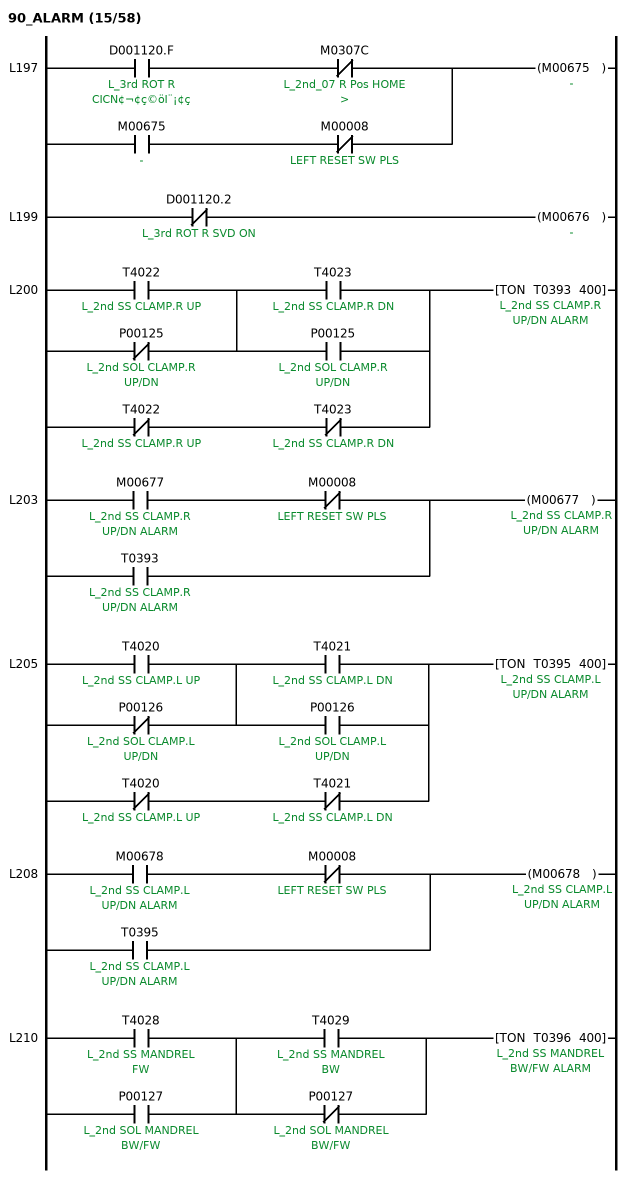
; L197
LOAD      D001120.F	// L_3rd ROT R CICN¢¬¢ç©öI¨¡¢ç
AND NOT   M0307C	// L_2nd_07 R Pos HOME >
LOAD      M00675	// -
AND NOT   M00008	// LEFT RESET SW PLS
OR LOAD
OUT       M00675	// -
; L199
LOAD NOT  D001120.2	// L_3rd ROT R SVD ON
OUT       M00676	// -
; L200
LOAD      T4022	// L_2nd SS CLAMP.R UP
OR NOT    P00125	// L_2nd SOL CLAMP.R UP/DN
LOAD      T4023	// L_2nd SS CLAMP.R DN
OR        P00125	// L_2nd SOL CLAMP.R UP/DN
AND LOAD
LOAD NOT  T4022	// L_2nd SS CLAMP.R UP
AND NOT   T4023	// L_2nd SS CLAMP.R DN
OR LOAD
TON       T0393 400	// L_2nd SS CLAMP.R UP/DN ALARM
; L203
LOAD      M00677	// L_2nd SS CLAMP.R UP/DN ALARM
AND NOT   M00008	// LEFT RESET SW PLS
OR        T0393	// L_2nd SS CLAMP.R UP/DN ALARM
OUT       M00677	// L_2nd SS CLAMP.R UP/DN ALARM
; L205
LOAD      T4020	// L_2nd SS CLAMP.L UP
OR NOT    P00126	// L_2nd SOL CLAMP.L UP/DN
LOAD      T4021	// L_2nd SS CLAMP.L DN
OR        P00126	// L_2nd SOL CLAMP.L UP/DN
AND LOAD
LOAD NOT  T4020	// L_2nd SS CLAMP.L UP
AND NOT   T4021	// L_2nd SS CLAMP.L DN
OR LOAD
TON       T0395 400	// L_2nd SS CLAMP.L UP/DN ALARM
; L208
LOAD      M00678	// L_2nd SS CLAMP.L UP/DN ALARM
AND NOT   M00008	// LEFT RESET SW PLS
OR        T0395	// L_2nd SS CLAMP.L UP/DN ALARM
OUT       M00678	// L_2nd SS CLAMP.L UP/DN ALARM
; L210
LOAD      T4028	// L_2nd SS MANDREL FW
OR        P00127	// L_2nd SOL MANDREL BW/FW
LOAD      T4029	// L_2nd SS MANDREL BW
OR NOT    P00127	// L_2nd SOL MANDREL BW/FW
AND LOAD
TON       T0396 400	// L_2nd SS MANDREL BW/FW ALARM

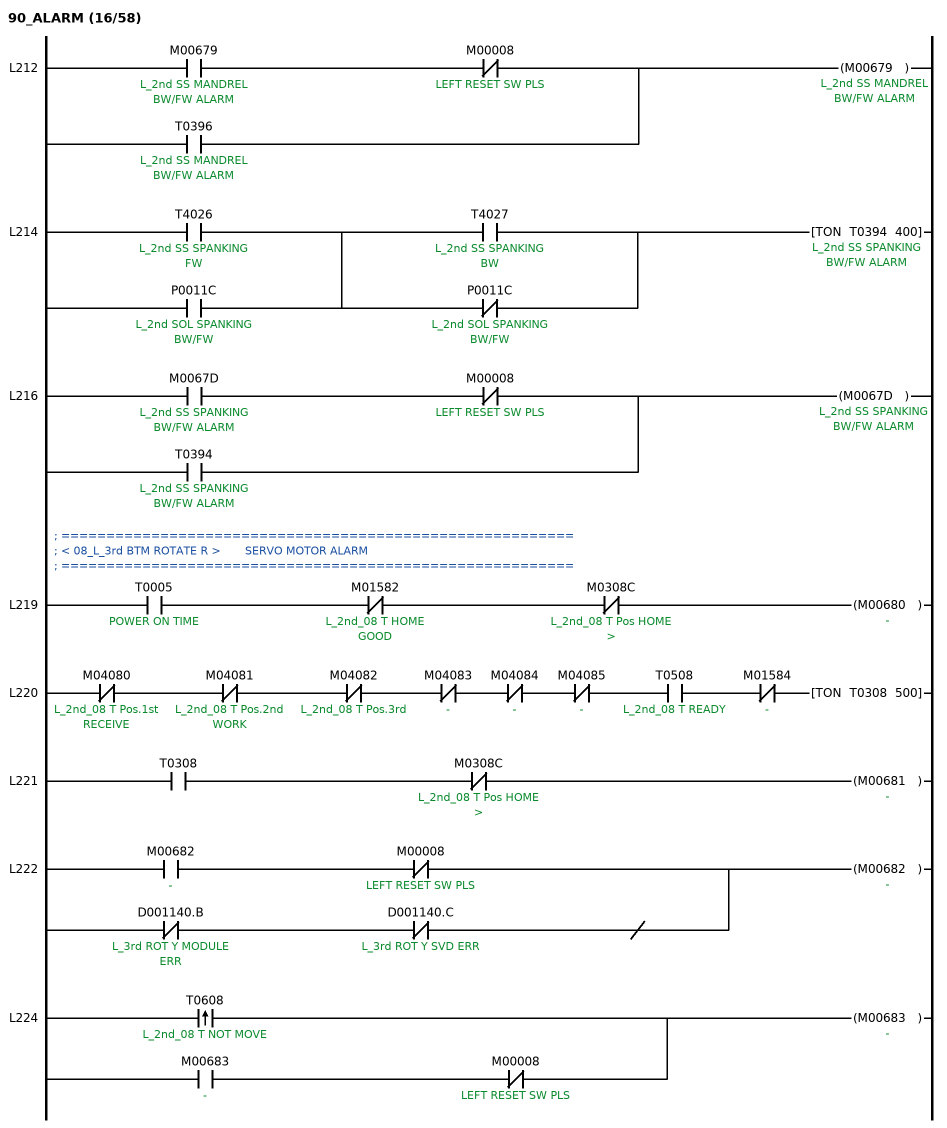
; L212
LOAD      M00679	// L_2nd SS MANDREL BW/FW ALARM
AND NOT   M00008	// LEFT RESET SW PLS
OR        T0396	// L_2nd SS MANDREL BW/FW ALARM
OUT       M00679	// L_2nd SS MANDREL BW/FW ALARM
; L214
LOAD      T4026	// L_2nd SS SPANKING FW
OR        P0011C	// L_2nd SOL SPANKING BW/FW
LOAD      T4027	// L_2nd SS SPANKING BW
OR NOT    P0011C	// L_2nd SOL SPANKING BW/FW
AND LOAD
TON       T0394 400	// L_2nd SS SPANKING BW/FW ALARM
; L216
LOAD      M0067D	// L_2nd SS SPANKING BW/FW ALARM
AND NOT   M00008	// LEFT RESET SW PLS
OR        T0394	// L_2nd SS SPANKING BW/FW ALARM
OUT       M0067D	// L_2nd SS SPANKING BW/FW ALARM
// =========================================================
// 
//        < 08_L_3rd BTM ROTATE R >       SERVO MOTOR ALARM
// 
// =========================================================
; L219
LOAD      T0005	// POWER ON TIME
AND NOT   M01582	// L_2nd_08 T HOME GOOD
AND NOT   M0308C	// L_2nd_08 T Pos HOME >
OUT       M00680	// -
; L220
LOAD NOT  M04080	// L_2nd_08 T Pos.1st RECEIVE
AND NOT   M04081	// L_2nd_08 T Pos.2nd WORK
AND NOT   M04082	// L_2nd_08 T Pos.3rd
AND NOT   M04083	// -
AND NOT   M04084	// -
AND NOT   M04085	// -
AND       T0508	// L_2nd_08 T READY
AND NOT   M01584	// -
TON       T0308 500
; L221
LOAD      T0308
AND NOT   M0308C	// L_2nd_08 T Pos HOME >
OUT       M00681	// -
; L222
LOAD      M00682	// -
AND NOT   M00008	// LEFT RESET SW PLS
LOAD NOT  D001140.B	// L_3rd ROT Y MODULE ERR
AND NOT   D001140.C	// L_3rd ROT Y SVD ERR
NOT
OR LOAD
OUT       M00682	// -
; L224
LOADP     T0608	// L_2nd_08 T NOT MOVE
LOAD      M00683	// -
AND NOT   M00008	// LEFT RESET SW PLS
OR LOAD
OUT       M00683	// -

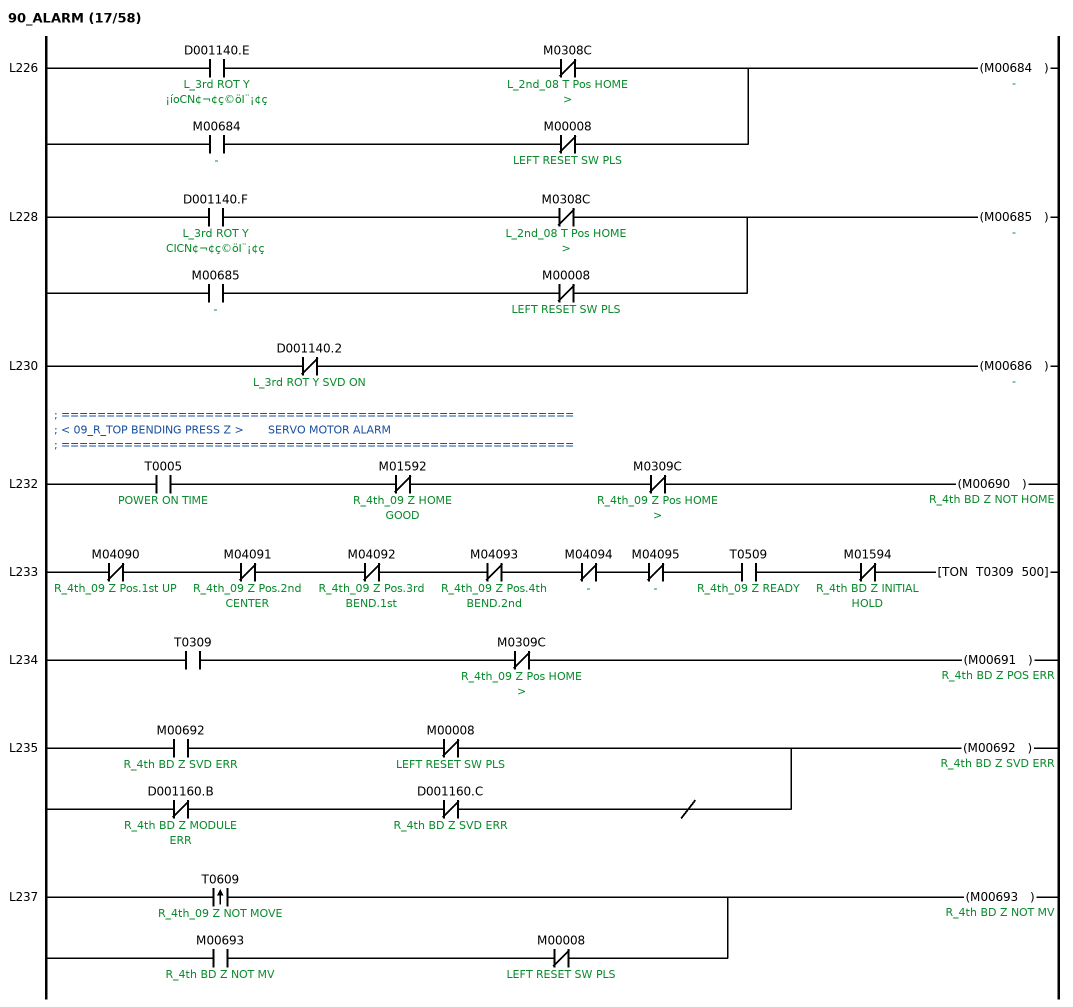
; L226
LOAD      D001140.E	// L_3rd ROT Y ¡íoCN¢¬¢ç©öI¨¡¢ç
AND NOT   M0308C	// L_2nd_08 T Pos HOME >
LOAD      M00684	// -
AND NOT   M00008	// LEFT RESET SW PLS
OR LOAD
OUT       M00684	// -
; L228
LOAD      D001140.F	// L_3rd ROT Y CICN¢¬¢ç©öI¨¡¢ç
AND NOT   M0308C	// L_2nd_08 T Pos HOME >
LOAD      M00685	// -
AND NOT   M00008	// LEFT RESET SW PLS
OR LOAD
OUT       M00685	// -
; L230
LOAD NOT  D001140.2	// L_3rd ROT Y SVD ON
OUT       M00686	// -
// =========================================================
// 
//        < 09_R_TOP BENDING PRESS Z >       SERVO MOTOR ALARM
// 
// =========================================================
; L232
LOAD      T0005	// POWER ON TIME
AND NOT   M01592	// R_4th_09 Z HOME GOOD
AND NOT   M0309C	// R_4th_09 Z Pos HOME >
OUT       M00690	// R_4th BD Z NOT HOME
; L233
LOAD NOT  M04090	// R_4th_09 Z Pos.1st UP
AND NOT   M04091	// R_4th_09 Z Pos.2nd CENTER
AND NOT   M04092	// R_4th_09 Z Pos.3rd BEND.1st
AND NOT   M04093	// R_4th_09 Z Pos.4th BEND.2nd
AND NOT   M04094	// -
AND NOT   M04095	// -
AND       T0509	// R_4th_09 Z READY
AND NOT   M01594	// R_4th BD Z INITIAL HOLD
TON       T0309 500
; L234
LOAD      T0309
AND NOT   M0309C	// R_4th_09 Z Pos HOME >
OUT       M00691	// R_4th BD Z POS ERR
; L235
LOAD      M00692	// R_4th BD Z SVD ERR
AND NOT   M00008	// LEFT RESET SW PLS
LOAD NOT  D001160.B	// R_4th BD Z MODULE ERR
AND NOT   D001160.C	// R_4th BD Z SVD ERR
NOT
OR LOAD
OUT       M00692	// R_4th BD Z SVD ERR
; L237
LOADP     T0609	// R_4th_09 Z NOT MOVE
LOAD      M00693	// R_4th BD Z NOT MV
AND NOT   M00008	// LEFT RESET SW PLS
OR LOAD
OUT       M00693	// R_4th BD Z NOT MV

